(* PLC project PLCC Raw Material Accounting System, Machine Expert Logic Builder V23.0.22.0, author nikiden *)
(* stored: creationDateTime 2026-09-22T13:28:06.869679+00:00, version 0.0.0.0, modificationDateTime 2026-09-10T08:01:48.8091995, organization Briansk Cardboard *)

TYPE E_ChannelStatus :
(
    CHANNEL_STATUS_STARTING     := 0,    // Ожидание первого корректного отсчёта HSC.
    CHANNEL_STATUS_RUNNING      := 1,    // Канал работает штатно.
    CHANNEL_STATUS_HSC_INVALID  := 2,    // HSC временно не подтверждает достоверность данных.
    CHANNEL_STATUS_HSC_ERROR    := 3,    // Аппаратный HSC сообщил об ошибке.
    CHANNEL_STATUS_COUNTER_JUMP := 4,    // Обнаружен недопустимо большой скачок счётчика.
    CHANNEL_STATUS_CONFIG_ERROR := 5     // Ошибка настроек диапазона HSC или пересчёта.
);
END_TYPE

TYPE E_RollEndReason :
(
    ROLL_END_NONE   := 0,    // Рулон ещё не завершался.
    ROLL_END_SPLICE := 1,    // Рулон завершён кнопкой SPLICE.
    ROLL_END_RESET  := 2     // Рулон завершён ручной кнопкой RESET.
);
END_TYPE

TYPE ST_HscState :
STRUCT
    xInitialized         : BOOL;             // Получен первый корректный абсолютный отсчёт HSC.
    udiPreviousAbs       : UDINT;            // Абсолютное значение HSC на предыдущем цикле.
    udiPulseDelta        : UDINT;            // Число новых импульсов за текущий цикл ПЛК.
    xDataValid           : BOOL;             // Приращение импульсов разрешено использовать.
    xJumpDetected        : BOOL;             // Одноцикловый признак недопустимого скачка HSC.
    udiRejectedJumpCount : UDINT;            // Количество отброшенных скачков HSC.
    eStatus              : E_ChannelStatus;  // Текущее состояние канала.
END_STRUCT
END_TYPE

TYPE ST_LineState :
STRUCT
    uliTotalPulses   : ULINT;  // Общее число импульсов шестого энкодера после запуска ПЛК.
    uliTotalLengthMm : ULINT;  // Общий метраж линии в миллиметрах после запуска ПЛК.
    rSpeedMPerMin    : REAL;   // Текущая скорость линии в метрах в минуту.
    xMoving          : BOOL;   // TRUE, если за последний интервал пришли импульсы.
    xConfigFault     : BOOL;   // Ошибка параметров энкодера, колеса или интервала скорости.
END_STRUCT
END_TYPE

TYPE ST_RollEvent :
STRUCT
    udiEventId         : UDINT;          // Уникальный номер события; назначается постоянной очередью.
    udiTimestampUtc    : UDINT;          // UNIX-время завершения рулона в секундах UTC.
    usiUnwindNumber    : USINT;          // Постоянный физический номер раската 1...5.
    usiShiftNumber     : USINT;          // Номер смены, в которой завершился рулон: 1 или 2.
    eEndReason         : E_RollEndReason;// Причина завершения: SPLICE или допустимый RESET.
    udiLengthMm        : UDINT;          // Итоговая длина завершённого рулона в миллиметрах, максимум около 4295 км.
END_STRUCT
END_TYPE

TYPE ST_RollState :
STRUCT
    uliCurrentRollPulses       : ULINT;           // Накопленные импульсы текущего рулона.
    uliCurrentLengthMm         : ULINT;           // Длина текущего рулона в миллиметрах.
    uliPreviousRollPulses      : ULINT;           // Импульсы последнего учтённого рулона.
    uliPreviousRollLengthMm    : ULINT;           // Длина последнего учтённого рулона в миллиметрах.
    udiRollSequenceNumber      : UDINT;           // Порядковый номер текущего рулона внутри канала.
    eLastEndReason             : E_RollEndReason; // Причина завершения предыдущего учтённого рулона.
    xRollCompleted             : BOOL;            // Одноцикловый сигнал завершения учтённого рулона.
    xShortResetDiscarded       : BOOL;            // Одноцикловый сигнал RESET при длине менее 100 м.
    uliLastDiscardedLengthMm   : ULINT;           // Длина последнего отброшенного короткого рулона.
    uliDiscardedTotalLengthMm  : ULINT;           // Общая отброшенная длина после коротких RESET.
    xConfigFault               : BOOL;            // Ошибка параметров энкодера или мерного колеса.
END_STRUCT
END_TYPE

TYPE ST_ShiftState :
STRUCT
    usiCurrentShift : USINT;  // Номер текущей смены: 1 или 2.
    xRtcValid       : BOOL;   // RTC контроллера прочитан без ошибки.
    xShiftChanged   : BOOL;   // Одноцикловый признак смены номера смены.
    uiLocalHour     : UINT;   // Текущий местный час, 0...23.
    uiLocalMinute   : UINT;   // Текущая местная минута, 0...59.
    uiLocalSecond   : UINT;   // Текущая местная секунда, 0...59.
    uiLocalYear     : UINT;   // Год местного времени, например 2026.
    uiLocalMonth    : UINT;   // Месяц местного времени, 1...12.
    uiLocalDay      : UINT;   // День месяца местного времени, 1...31.
    udiTimestampUtc : UDINT;  // Текущее UNIX-время в секундах UTC для отметки событий.
    udiRtcError     : UDINT;  // Код ошибки функции чтения RTC, 0 означает отсутствие ошибки.
END_STRUCT
END_TYPE

TYPE ST_StopJournalEvent :
STRUCT
    udiEventId                  : UDINT; // Постоянный ID события линии ЛГК.
    udiTimestampUtc             : UDINT; // UNIX UTC; 0, если RTC неисправен.
    wKind                       : WORD;  // 1=состояние, 2=завершение смены, 3=новый заказ.
    wStateCode                  : WORD;  // Старые коды ProductionLine; 32768=граница смены.
    wShiftNumber                : WORD;  // Смена, к которой относится снимок.
    udiOrderNumber              : UDINT; // Номер заказа на момент события.
    udiOrderLengthDm            : UDINT; // Метраж заказа, 0,1 м.
    udiOrderAreaX100            : UDINT; // Площадь заказа, м2 x 100.
    udiShiftLengthDm            : UDINT; // Метраж смены, 0,1 м.
    udiShiftAreaX100            : UDINT; // Площадь смены, м2 x 100.
    wSpeedDmPerMin              : WORD;  // Скорость, 0,1 м/мин.
    wOperatorNumber             : WORD;  // Номер оператора.
    wChangeoverSetpointTenthsMin: WORD;  // Норматив переналадки, 0,1 мин.
    wAlarmBits                  : WORD;  // Диагностика нового ПЛК; не старый Status2.
    wBreakPoint                 : WORD;  // Точка обрыва 1...5.
    wBreakSide                  : WORD;  // Сторона обрыва 1...2.
    wBreakReason                : WORD;  // Причина обрыва 1...3.
END_STRUCT
END_TYPE

TYPE ST_StopJournalPersistent :
STRUCT
    a_stQueue        : ARRAY[0..127] OF ST_StopJournalEvent;
    uiHead           : UINT;
    uiTail           : UINT;
    uiCount          : UINT;
    udiNextEventId   : UDINT;
    udiOverflowCount : UDINT;
    uliLinePulses    : ULINT;
    wLastState       : WORD;
    dwSignature      : DWORD;
END_STRUCT
END_TYPE

TYPE ST_StopMachinePersistent :
STRUCT
    wConfigSignature                 : WORD;  // Сигнатура инициализированных постоянных настроек.
    udiOrderNumber                   : UDINT; // Номер заказа, показываемый оператору.
    udiOrderDatabaseId               : UDINT; // NumZ: ключ записи заказа в БД.
    udiOrderTechnicalCard            : UDINT; // NumTK: номер технологической карты.
    uiOrderSourceShift               : UINT;  // NumSM, полученный с сервера.
    uiOrderNominalSpeed              : UINT;  // Efficiency из записи заказа.
    uiOperatorNumber                 : UINT;  // Номер авторизованного оператора будущей EB-панели.
    wLastServerOrderSequence         : WORD;  // Последний атомарно применённый пакет сервера.
    uliOrderBaselineMm               : ULINT; // Общий метраж линии в момент начала заказа.
    uliShiftBaselineMm               : ULINT; // Общий метраж линии в момент начала смены.
    uiAreaCoefficientX100            : UINT;  // Площадь на метр, м2/м x 100 (210 = 2,10).
    uiStartDetectLengthDm            : UINT;  // Путь подтверждения работы, 0,1 м.
    uiChangeoverSetpointTenthsMin    : UINT;  // Допустимая переналадка, 0,1 мин.
    usiLastShiftNumber               : USINT; // Последняя смена для восстановления после отключения.
END_STRUCT
END_TYPE

TYPE ST_StopMachineState :
STRUCT
    wStateCode                         : WORD;  // Текущее состояние ЛГК по таблице состояний.
    wStatusBits                        : WORD;  // Диагностические признаки интерфейса Стопмашины.
    wAlarmBits                         : WORD;  // Активные предупреждения интерфейса.
    udiOrderNumber                     : UDINT; // Номер текущего заказа.
    udiOrderDatabaseId                 : UDINT; // Ключ текущего заказа в БД.
    udiOrderTechnicalCard              : UDINT; // Номер технологической карты.
    uiOrderSourceShift                 : UINT;  // Номер смены из записи заказа сервера.
    uiOrderNominalSpeed                : UINT;  // Номинальная скорость из записи заказа.
    uiOperatorNumber                   : UINT;  // Номер оператора EB-панели.
    udiCurrentOrderLengthDm            : UDINT; // Выпуск текущего заказа, 0,1 м.
    udiShiftLengthDm                   : UDINT; // Выпуск текущей смены, 0,1 м.
    udiCurrentOrderAreaX100            : UDINT; // Площадь текущего заказа, м2 x 100.
    udiShiftAreaX100                   : UDINT; // Площадь текущей смены, м2 x 100.
    uiSpeedDmPerMin                    : UINT;  // Скорость, 0,1 м/мин.
    uiChangeoverRemainingTenthsMin     : UINT;  // Остаток переналадки, 0,1 мин.
    usiLastBreakPoint                  : USINT; // Последняя точка обрыва: 1...5.
    usiLastBreakSide                   : USINT; // Сторона: 1 верх, 2 низ.
    usiLastBreakReason                 : USINT; // Причина: 1 сырьё, 2 оборудование, 3 машинист.
    wLastCommandResult                 : WORD;  // Результат последней обработанной команды HMI.
    wLastProcessedSequence             : WORD;  // Последовательность последней команды HMI.
    wLastServerOrderResult              : WORD;  // Результат обработки последнего пакета заказа.
    wLastServerOrderSequence            : WORD;  // Последовательность последнего пакета заказа.
    xPackingComplete                   : BOOL;  // Оператор подтвердил завершение упаковки.
    xChangeoverOverdue                 : BOOL;  // Превышено заданное время переналадки.
    xCommandRejected                   : BOOL;  // Последняя полученная команда отклонена.
    xConfigFault                       : BOOL;  // Некорректные сохранённые настройки.
    xServerOrderValid                  : BOOL;  // PLC получил корректный заказ от сервера.
    xInitialized                       : BOOL;  // Блок прошёл первичную инициализацию.
END_STRUCT
END_TYPE

TYPE ST_SystemDiagnostics :
STRUCT
    a_eHscStatus      : ARRAY[1..6] OF E_ChannelStatus; // Состояния шести каналов HSC.
    a_xHscFault       : ARRAY[1..6] OF BOOL;            // Ошибка соответствующего канала HSC.
    a_xHmiOverflow    : ARRAY[1..5] OF BOOL;            // Значение канала не помещается в 32 бита DWIN.
    xAnyHscFault      : BOOL;                           // Есть хотя бы одна ошибка HSC.
    xAnyConfigFault   : BOOL;                           // Есть ошибка параметров пересчёта.
    xRtcFault         : BOOL;                           // Не удалось получить время контроллера.
    uliProgramCycles  : ULINT;                          // Счётчик циклов SR_Main для диагностики.
END_STRUCT
END_TYPE

(* global variable list GVL_Constants *)
VAR_GLOBAL CONSTANT
    c_iRollChannelCount              : INT   := 5;                    // Количество раскатов сырья.
    c_iHscChannelCount               : INT   := 6;                    // Пять раскатов и один энкодер линии.
    c_udiEncoderPulsesPerRevolution  : UDINT := UDINT#250;            // Импульсов энкодера за один оборот.
    c_udiWheelCircumferenceMm        : UDINT := UDINT#250;            // Окружность каждого мерного колеса, мм.
    c_udiHscCounterRange             : UDINT := UDINT#1000000000;     // Диапазон HSC: значения 0...999999999.
    c_udiMaxPulseDeltaPerCycle       : UDINT := UDINT#100000;         // Защита от ложного скачка или сброса HSC.
    c_tInputFilter                   : TIME  := T#50ms;                // Время подтверждения нажатия кнопки.
    c_uliManualResetMinLengthMm      : ULINT := ULINT#100000;         // Минимум 100 м для учёта ручного RESET.
    c_tSpeedSample                   : TIME  := T#1s;                  // Интервал обновления скорости линии.
    c_tHaiwellActivityHold           : TIME  := T#10s;                 // Удержание признака движения для медленного опроса HMI.
    c_tHaiwellFlashHalfPeriod        : TIME  := T#250ms;               // Три быстрые жёлтые вспышки: 0,25 с ВКЛ и 0,25 с ВЫКЛ.
    c_tHaiwellResetHold              : TIME  := T#3s;                  // Время показа состояния RESET на центральной HMI.
    c_usiShift_1_StartHour           : USINT := USINT#8;              // Начало первой смены, 08:00.
    c_usiShift_2_StartHour           : USINT := USINT#20;             // Начало второй смены, 20:00.
    c_udiShiftMaxIntervalSeconds     : UDINT := UDINT#43200;          // Максимум одного сменного интервала: 12 часов.
    c_udiLocalUtcOffsetSeconds       : UDINT := UDINT#10800;          // Брянск: UTC+3, то есть 3 часа.
    c_dwPersistentLayoutSignature    : DWORD := DWORD#16#4342504C;    // ASCII "CBPL": признак нашей структуры PERSISTENT.
    c_wPersistentLayoutVersion       : WORD  := WORD#2;                // Версия разметки постоянной памяти.
    c_wHaiwellProtocolVersion        : WORD  := WORD#2;                // Версия read-only карты центральной Haiwell.

    // Отдельный интерфейс Стопмашины ЛГК. Он не содержит номера линии.
    c_wStopMachineSignature          : WORD  := WORD#16#534D;         // ASCII "SM".
    c_wStopMachineProtocolVersion    : WORD  := WORD#2;
    c_wServerOrderApplyCommand       : WORD  := WORD#16#4F52;         // ASCII "OR": применить пакет заказа сервера.
    c_uiStopDefaultAreaCoefficientX100 : UINT := UINT#210;            // 2,10 м2 на метр.
    c_uiStopDefaultStartDetectLengthDm : UINT := UINT#500;            // 50,0 м.
    c_uiStopDefaultChangeoverTenthsMin : UINT := UINT#0;              // Таймер отключён до настройки.
    c_tStopNoFeedDelay               : TIME  := T#20s;

    c_wStopStateRunning              : WORD := WORD#1;
    c_wStopStateStopped              : WORD := WORD#2;
    c_wStopStateNoFeed               : WORD := WORD#8;
    c_wStopStateChangeover           : WORD := WORD#16;
    c_wStopStateProduction           : WORD := WORD#32;
    c_wStopStatePpr                  : WORD := WORD#64;
    c_wStopStateLunch                : WORD := WORD#128;
    c_wStopStateRepair               : WORD := WORD#256;
    c_wStopStateAlarm                : WORD := WORD#512;
    c_wStopStateTechnology           : WORD := WORD#1024;
    c_wStopStateBreak                : WORD := WORD#2048;

    c_wStopCommandStop               : WORD := WORD#1;
    c_wStopCommandStart              : WORD := WORD#2;
    c_wStopCommandChangeover         : WORD := WORD#3;
    c_wStopCommandProduction         : WORD := WORD#4;
    c_wStopCommandLunch              : WORD := WORD#5;
    c_wStopCommandPpr                : WORD := WORD#6;
    c_wStopCommandRepair             : WORD := WORD#7;
    c_wStopCommandAlarm              : WORD := WORD#8;
    c_wStopCommandTechnology         : WORD := WORD#9;
    c_wStopCommandBreak              : WORD := WORD#10;
    c_wStopCommandPackingComplete    : WORD := WORD#11;
    c_wStopCommandSetOperator        : WORD := WORD#12;
    c_wStopCommandApplySettings      : WORD := WORD#20;

    c_wStopResultNone                : WORD := WORD#0;
    c_wStopResultAccepted            : WORD := WORD#1;
    c_wStopResultInvalidCode         : WORD := WORD#2;
    c_wStopResultInvalidParameter    : WORD := WORD#3;
    c_wStopResultInvalidState        : WORD := WORD#4;                // Команда состояния противоречит движению энкодера.
END_VAR

(* global variable list GVL_IO *)
VAR_GLOBAL
    udiHscAbs : ARRAY[1..6] OF UDINT; // Абсолютные показания шести аппаратных HSC.
    xHscValid : ARRAY[1..6] OF BOOL;  // Достоверность выходов соответствующего HSC.
    xHscError : ARRAY[1..6] OF BOOL;  // Ошибка соответствующего аппаратного HSC.
    xReset    : ARRAY[1..5] OF BOOL;  // Кнопки RESET раскатов 1...5 с TM3DI16, входы I0...I4.
    xSplice   : ARRAY[1..5] OF BOOL;  // Кнопки SPLICE раскатов 1...5 с TM3DI16, входы I5...I9.
END_VAR

(* global variable list GVL_Runtime *)
VAR_GLOBAL
    a_stHscState  : ARRAY[1..6] OF ST_HscState;  // Рабочее состояние шести каналов HSC.
    stLineState   : ST_LineState;                // Скорость и общий метраж шестого энкодера.
    stShiftState  : ST_ShiftState;               // Номер смены и состояние часов контроллера.
    stStopMachine : ST_StopMachineState;         // Изолированное состояние Стопмашины линии ЛГК.
END_VAR

(* global variable list GVL_HMI *)
VAR_GLOBAL
    a_wHmi1Tx : ARRAY[0..12] OF WORD; // Регистры VP 2000...200C панели раската №1.
    a_wHmi2Tx : ARRAY[0..12] OF WORD; // Регистры VP 2000...200C панели раската №2.
    a_wHmi3Tx : ARRAY[0..12] OF WORD; // Регистры VP 2000...200C панели раската №3.
    a_wHmi4Tx : ARRAY[0..12] OF WORD; // Регистры VP 2000...200C панели раската №4.
    a_wHmi5Tx : ARRAY[0..12] OF WORD; // Регистры VP 2000...200C панели раската №5.

    // Системный пакет установки встроенных часов DWIN через VP 009C...009F.
    a_wHmi1RtcSync : ARRAY[0..3] OF WORD;
    a_wHmi2RtcSync : ARRAY[0..3] OF WORD;
    a_wHmi3RtcSync : ARRAY[0..3] OF WORD;
    a_wHmi4RtcSync : ARRAY[0..3] OF WORD;
    a_wHmi5RtcSync : ARRAY[0..3] OF WORD;
END_VAR

(* global variable list GVL_Diagnostics *)
VAR_GLOBAL
    stSystem : ST_SystemDiagnostics; // Общая диагностика проекта для онлайн-контроля и будущей SCADA.
END_VAR

(* global variable list PersistentVars *)
VAR_GLOBAL PERSISTENT RETAIN
    a_stEventQueue       : ARRAY[0..127] OF ST_RollEvent; // Постоянная кольцевая очередь на 128 событий.
    uiEventQueueHead     : UINT := UINT#0;                // Индекс первого события, ожидающего подтверждения.
    uiEventQueueTail     : UINT := UINT#0;                // Индекс ячейки для записи следующего события.
    uiEventQueueCount    : UINT := UINT#0;                // Текущее количество событий в очереди.
    udiNextEventId       : UDINT := UDINT#1;              // Уникальный номер, который получит следующее событие.
    udiQueueOverflowCount: UDINT := UDINT#0;              // Число событий, не помещённых из-за полной очереди.
    a_stRollState        : ARRAY[1..5] OF ST_RollState;   // Сохраняемое состояние текущего и предыдущего рулона каждого раската.
    stStopMachine        : ST_StopMachinePersistent;      // Заказ, базовые метражи и настройки Стопмашины ЛГК.
    usiShiftAccumulatorNumber : USINT;                    // Смена, к которой относятся накопители центральной HMI.
    udiShiftStartTimestampUtc : UDINT;                    // UTC-время начала текущего интервала накопления.
    a_uliShiftRollPulses : ARRAY[1..5] OF ULINT;           // Импульсы каждого раската с начала текущей смены.
    uliShiftOutputPulses : ULINT;                          // Импульсы шестого энкодера с начала текущей смены.
    dwLayoutSignature    : DWORD;                          // Сигнатура разметки; ноль или несовпадение запускает безопасную инициализацию.
    wLayoutVersion       : WORD;                           // Версия разметки постоянной памяти.
    stStopJournal        : ST_StopJournalPersistent;       // Независимая очередь событий ЛГК; добавлена в конец разметки.
END_VAR

(* global variable list GVL_SCADA *)
VAR_GLOBAL
    a_wEventPacket AT %MW2000 : ARRAY[0..11] OF WORD; // Событие протокола v2: 12 последовательных слов.
    wEventReady AT %MW2012 : WORD;                    // 1 — пакет содержит событие, 0 — очередь пуста.
    wQueueCount AT %MW2013 : WORD;                    // Количество неподтверждённых событий в очереди.
    wQueueCapacity AT %MW2014 : WORD;                 // Полная ёмкость очереди, сейчас 128 событий.
    wQueueStatus AT %MW2015 : WORD;                   // 0 — пусто, 1 — есть данные, 2 — заполнена, 3 — ошибка хранилища, 4 — исчерпан EventId.

    a_wAckEventId AT %MW2016 : ARRAY[0..1] OF WORD;   // EventId UDINT, подтверждаемый сервером; старшее слово первым.
    wAckCommand AT %MW2018 : WORD;                    // Сервер записывает 16#A55A после сохранения события на диск.
    wCollectorHeartbeat AT %MW2019 : WORD;            // Счётчик жизни службы-сборщика; записывается сервером.
    wLastAckResult AT %MW2020 : WORD;                 // 0 — подтверждений не было, 1 — принято, 2 — отклонено.
    a_wQueueOverflowCount AT %MW2021 : ARRAY[0..1] OF WORD; // Число событий, отвергнутых из-за полной очереди.

    // Сервер -> PLC: новый заказ ЛГК. Параметры и sequence записываются первыми,
    // wOrderCommand = 16#4F52 записывается последним. PLC очищает команду сам.
    wOrderCommand AT %MW2030 : WORD;
    wOrderSequence AT %MW2031 : WORD;
    a_wOrderDatabaseId AT %MW2032 : ARRAY[0..1] OF WORD;     // NumZ из ExternalProductionData, старшее слово первым.
    a_wOrderTechnicalCard AT %MW2034 : ARRAY[0..1] OF WORD;  // NumTK, старшее слово первым.
    a_wOrderDisplayNumber AT %MW2036 : ARRAY[0..1] OF WORD;  // Числовая часть Zakaz для экрана, старшее слово первым.
    wOrderSourceShift AT %MW2038 : WORD;                     // NumSM от сервера.
    wOrderNominalSpeed AT %MW2039 : WORD;                    // Efficiency, единицы исходной БД.
    wOrderChangeoverTenthsMin AT %MW2040 : WORD;             // ReconfigurationT x 10.

    // PLC -> сервер: результат применения заказа.
    wOrderApplyResult AT %MW2041 : WORD;                     // 0 — нет, 1 — принят, 2 — неверная команда, 3 — неверные данные.
    wLastOrderSequence AT %MW2042 : WORD;
END_VAR

(* global variable list GVL_HAIWELL *)
VAR_GLOBAL
    // Непрерывная read-only область Modbus TCP для центральной Haiwell A10-W.
    // Многословные значения передаются в порядке: старшее WORD, затем младшее WORD.

    wHmiSignature       AT %MW2100 : WORD; // 16#484D ('HM').
    wHmiProtocolVersion AT %MW2101 : WORD; // Версия карты.
    wPlcHeartbeat       AT %MW2102 : WORD; // Изменяется раз в секунду.
    wSystemStatusBits   AT %MW2103 : WORD; // Общие диагностические флаги.
    wCurrentShift       AT %MW2104 : WORD; // 1, 2 или 0 при недостоверном RTC.
    wLocalHour          AT %MW2105 : WORD; // 0...23.
    wLocalMinute        AT %MW2106 : WORD; // 0...59.
    wEventQueueCount    AT %MW2107 : WORD;
    wEventQueueStatus   AT %MW2108 : WORD;
    wLastAckResult      AT %MW2109 : WORD;

    a_wCurrentLengthX10  AT %MW2110 : ARRAY[1..5, 0..1] OF WORD;
    a_wPreviousLengthX10 AT %MW2120 : ARRAY[1..5, 0..1] OF WORD;
    a_wUnwindStatus      AT %MW2130 : ARRAY[1..5] OF WORD;
    a_wLastEndReason     AT %MW2135 : ARRAY[1..5] OF WORD;

    a_wOutputTotalLengthX10 AT %MW2140 : ARRAY[0..1] OF WORD;
    wOutputSpeedX10         AT %MW2142 : WORD;
    wOutputStatus           AT %MW2143 : WORD;
    a_wDiscardedLengthX10   AT %MW2144 : ARRAY[1..5, 0..1] OF WORD;
    a_wQueueOverflowCount   AT %MW2154 : ARRAY[0..1] OF WORD;
    wCollectorHeartbeat     AT %MW2156 : WORD;
    wReserved2157           AT %MW2157 : WORD;

    // Состояния, дата и накопители текущей смены.
    a_wUnwindDisplayState       AT %MW2200 : ARRAY[1..5] OF WORD;    // 0 — стоит, 1 — работает, 2 — жёлтая фаза SPLICE/RESET.
    wLocalYear                  AT %MW2205 : WORD;
    wLocalMonth                 AT %MW2206 : WORD;
    wLocalDay                   AT %MW2207 : WORD;
    a_wReserved2208             AT %MW2208 : ARRAY[0..1] OF WORD;
    a_wShiftOutputLengthX10     AT %MW2210 : ARRAY[0..1] OF WORD;
    wShiftAverageSpeedX10       AT %MW2212 : WORD;
    wShiftStatus                AT %MW2213 : WORD;                   // bit 0 — накопители достоверны.
    a_wShiftRollLengthX10       AT %MW2214 : ARRAY[1..5, 0..1] OF WORD;
    a_wShiftRawTotalLengthX10   AT %MW2224 : ARRAY[0..1] OF WORD;
    a_wReserved2226             AT %MW2226 : ARRAY[0..3] OF WORD;
END_VAR

(* global variable list GVL_StopMachine *)
VAR_GLOBAL
    // ========================================================
    // PLC -> HMI. Только чтение со стороны панели, MW2300...2359
    // ========================================================
    wSignature AT %MW2300 : WORD;
    wProtocolVersion AT %MW2301 : WORD;
    wPlcHeartbeat AT %MW2302 : WORD;
    wStateCode AT %MW2303 : WORD;
    wStatusBits AT %MW2304 : WORD;
    wAlarmBits AT %MW2305 : WORD;
    wShiftNumber AT %MW2306 : WORD;
    wLocalHour AT %MW2307 : WORD;
    wLocalMinute AT %MW2308 : WORD;
    wLocalSecond AT %MW2309 : WORD;
    a_wOrderNumber AT %MW2310 : ARRAY[0..1] OF WORD;
    a_wOrderLengthDm AT %MW2312 : ARRAY[0..1] OF WORD;
    a_wOrderAreaX100 AT %MW2314 : ARRAY[0..1] OF WORD;
    a_wShiftLengthDm AT %MW2316 : ARRAY[0..1] OF WORD;
    a_wShiftAreaX100 AT %MW2318 : ARRAY[0..1] OF WORD;
    wSpeedDmPerMin AT %MW2320 : WORD;
    wChangeoverRemainingTenthsMin AT %MW2321 : WORD;
    wChangeoverSetpointTenthsMin AT %MW2322 : WORD;
    wStartDetectLengthDm AT %MW2323 : WORD;
    wAreaCoefficientX100 AT %MW2324 : WORD;
    wLastBreakPoint AT %MW2325 : WORD;
    wLastBreakSide AT %MW2326 : WORD;
    wLastBreakReason AT %MW2327 : WORD;
    wPackingComplete AT %MW2328 : WORD;
    wLastCommandResult AT %MW2329 : WORD;
    wLastProcessedSequence AT %MW2330 : WORD;
    wPhysicalControlEnabled AT %MW2331 : WORD; // Всегда 0: HMI не управляет оборудованием.
    a_wOrderDatabaseId AT %MW2332 : ARRAY[0..1] OF WORD;
    a_wOrderTechnicalCard AT %MW2334 : ARRAY[0..1] OF WORD;
    wOrderSourceShift AT %MW2336 : WORD;
    wOrderNominalSpeed AT %MW2337 : WORD;
    wOperatorNumber AT %MW2338 : WORD;
    a_wReservedRead AT %MW2339 : ARRAY[0..20] OF WORD;

    // ========================================================
    // HMI -> PLC. Панель пишет только MW2360...2399
    // Команда передаётся последней; sequence меняется для каждого действия.
    // ========================================================
    wCommandCode AT %MW2360 : WORD;
    wCommandSequence AT %MW2361 : WORD;
    wCommandParam0 AT %MW2362 : WORD;
    wCommandParam1 AT %MW2363 : WORD;
    wCommandParam2 AT %MW2364 : WORD;
    wSettingStartDetectLengthDm AT %MW2365 : WORD;
    wSettingAreaCoefficientX100 AT %MW2366 : WORD;
    wSettingChangeoverTenthsMin AT %MW2367 : WORD;
    wHmiHeartbeat AT %MW2368 : WORD;
    a_wReservedWrite AT %MW2369 : ARRAY[0..30] OF WORD;
END_VAR

(* global variable list GVL_StopJournal *)
VAR_GLOBAL
    // Снимок первого события. PLC -> сервер, 2400...2422.
    wSignature AT %MW2400 : WORD;                 // 16#534A = SJ.
    wVersion AT %MW2401 : WORD;                   // Версия протокола 1.
    a_wEventId AT %MW2402 : ARRAY[0..1] OF WORD; // Старшее слово первым.
    a_wTimestampUtc AT %MW2404 : ARRAY[0..1] OF WORD;
    wKind AT %MW2406 : WORD;
    wStateCode AT %MW2407 : WORD;
    wShiftNumber AT %MW2408 : WORD;
    a_wOrderNumber AT %MW2409 : ARRAY[0..1] OF WORD;
    a_wOrderLengthDm AT %MW2411 : ARRAY[0..1] OF WORD;
    a_wOrderAreaX100 AT %MW2413 : ARRAY[0..1] OF WORD;
    wSpeedDmPerMin AT %MW2415 : WORD;
    wOperatorNumber AT %MW2416 : WORD;
    wChangeoverSetpointTenthsMin AT %MW2417 : WORD;
    wAlarmBits AT %MW2418 : WORD;
    wBreakPoint AT %MW2419 : WORD;
    wBreakSide AT %MW2420 : WORD;
    wBreakReason AT %MW2421 : WORD;
    a_wShiftLengthDm AT %MW2422 : ARRAY[0..1] OF WORD;
    a_wShiftAreaX100 AT %MW2424 : ARRAY[0..1] OF WORD;
    wEventReady AT %MW2426 : WORD;
    wQueueCount AT %MW2427 : WORD;
    wQueueStatus AT %MW2428 : WORD;               // 0=норма, 1=полна, 2=переполнение, 3=повреждение, 4=ID исчерпан.
    // Сервер -> PLC: ID записать первым, команду 16#A55B — последней.
    a_wAckEventId AT %MW2429 : ARRAY[0..1] OF WORD;
    wAckCommand AT %MW2431 : WORD;
    wLastAckResult AT %MW2432 : WORD;             // 0=нет, 1=принят, 2=отклонён.
    a_wOverflowCount AT %MW2433 : ARRAY[0..1] OF WORD;
    wHeartbeat AT %MW2435 : WORD;
    a_wReserved AT %MW2436 : ARRAY[0..23] OF WORD;
END_VAR

FUNCTION_BLOCK FB_DwinDataPacker
VAR_INPUT
    i_uliCurrentLengthMm  : ULINT; // Текущая длина рулона в миллиметрах.
    i_uliPreviousLengthMm : ULINT; // Предыдущая длина рулона в миллиметрах.
    i_usiUnwindNumber     : USINT; // Постоянный физический номер раската 1...5.
END_VAR

VAR_OUTPUT
    q_wCurrentHigh  : WORD; // VP 2000: старшее слово текущей длины.
    q_wCurrentLow   : WORD; // VP 2001: младшее слово текущей длины.
    q_wPreviousHigh : WORD; // VP 2002: старшее слово предыдущей длины.
    q_wPreviousLow  : WORD; // VP 2003: младшее слово предыдущей длины.
    q_wUnwindNumber : WORD; // VP 2004: постоянный физический номер раската.
    q_xOverflow     : BOOL; // Одно из значений превысило диапазон 32-битного DWIN.
END_VAR

VAR
    uliCurrentX10  : ULINT; // Текущая длина в десятых долях метра.
    uliPreviousX10 : ULINT; // Предыдущая длина в десятых долях метра.
    udiCurrentX10  : UDINT; // Ограниченное 32-битное значение текущей длины.
    udiPreviousX10 : UDINT; // Ограниченное 32-битное значение предыдущей длины.
END_VAR

VAR CONSTANT
    c_uliDwinMaxValue : ULINT := ULINT#4294967295; // Максимум Unsigned Long Int DWIN.
END_VAR

            // 100 мм соответствуют 0.1 м на экране DWIN.
uliCurrentX10 := i_uliCurrentLengthMm / ULINT#100;
uliPreviousX10 := i_uliPreviousLengthMm / ULINT#100;
IF (i_uliPreviousLengthMm MOD ULINT#100) >= ULINT#50 THEN
    uliPreviousX10 := uliPreviousX10 + ULINT#1;
END_IF;
q_xOverflow := FALSE;


IF uliCurrentX10 > c_uliDwinMaxValue THEN
    udiCurrentX10 := UDINT#4294967295;
    q_xOverflow := TRUE;
ELSE
    udiCurrentX10 := ULINT_TO_UDINT(uliCurrentX10);
END_IF;


IF uliPreviousX10 > c_uliDwinMaxValue THEN
    udiPreviousX10 := UDINT#4294967295;
    q_xOverflow := TRUE;
ELSE
    udiPreviousX10 := ULINT_TO_UDINT(uliPreviousX10);
END_IF;


q_wCurrentHigh :=
    UDINT_TO_WORD(udiCurrentX10 / UDINT#65536);

q_wCurrentLow :=
    UDINT_TO_WORD(udiCurrentX10 MOD UDINT#65536);

q_wPreviousHigh :=
    UDINT_TO_WORD(udiPreviousX10 / UDINT#65536);

q_wPreviousLow :=
    UDINT_TO_WORD(udiPreviousX10 MOD UDINT#65536);

q_wUnwindNumber := USINT_TO_WORD(i_usiUnwindNumber);

          
END_FUNCTION_BLOCK

FUNCTION_BLOCK FB_EventPacker
VAR_INPUT
    i_xEventValid : BOOL;         // TRUE — входная структура содержит событие для передачи.
    i_stEvent     : ST_RollEvent; // Первое неподтверждённое событие постоянной очереди.
END_VAR

VAR_OUTPUT
    q_a_wPacket   : ARRAY[0..11] OF WORD; // Пакет протокола v2: 12 слов, старшие слова идут первыми.
    q_xPacketValid: BOOL;                 // TRUE — пакет заполнен и CRC рассчитан.
END_VAR

VAR
    iWord       : INT;  // Индекс слова при очистке пакета и вычислении CRC.
    iByte       : INT;  // Индекс байта внутри слова: сначала старший, затем младший.
    iBit        : INT;  // Индекс бита при вычислении CRC16 Modbus.
    wCrc        : WORD; // Рабочее значение CRC16 Modbus.
    wSourceWord : WORD; // Текущее слово пакета, участвующее в CRC.
    byData      : BYTE; // Текущий байт пакета, участвующий в CRC.
END_VAR

VAR CONSTANT
    c_wSignature      : WORD := WORD#16#CB01; // Сигнатура протокола CBPL, защищает от неверного разбора пакета.
    c_wProtocolVersion: WORD := WORD#2;       // Версия 2: EventId и длина передаются как UDINT.
END_VAR

            q_xPacketValid := FALSE;

FOR iWord := 0 TO 11 DO
    q_a_wPacket[iWord] := WORD#0;
END_FOR;


IF i_xEventValid THEN

    // 0: сигнатура; 1: версия протокола.
    q_a_wPacket[0] := c_wSignature;
    q_a_wPacket[1] := c_wProtocolVersion;

    // 2...3: EventId UDINT, старшее слово идёт первым.
    q_a_wPacket[2] := UDINT_TO_WORD(i_stEvent.udiEventId / UDINT#65536);
    q_a_wPacket[3] := UDINT_TO_WORD(i_stEvent.udiEventId MOD UDINT#65536);

    // 4...5: UNIX-время UTC UDINT, старшее слово идёт первым.
    q_a_wPacket[4] := UDINT_TO_WORD(i_stEvent.udiTimestampUtc / UDINT#65536);
    q_a_wPacket[5] := UDINT_TO_WORD(i_stEvent.udiTimestampUtc MOD UDINT#65536);

    // 6...8: физический раскат, смена и причина передаются отдельными словами.
    q_a_wPacket[6] := USINT_TO_WORD(i_stEvent.usiUnwindNumber);
    q_a_wPacket[7] := USINT_TO_WORD(i_stEvent.usiShiftNumber);

    CASE i_stEvent.eEndReason OF
        ROLL_END_SPLICE:
            q_a_wPacket[8] := WORD#1;
        ROLL_END_RESET:
            q_a_wPacket[8] := WORD#2;
        ELSE
            q_a_wPacket[8] := WORD#0;
    END_CASE;

    // 9...10: длина завершённого рулона в миллиметрах, UDINT.
    q_a_wPacket[9] := UDINT_TO_WORD(i_stEvent.udiLengthMm / UDINT#65536);
    q_a_wPacket[10] := UDINT_TO_WORD(i_stEvent.udiLengthMm MOD UDINT#65536);


    // CRC16 Modbus по словам 0...10. В каждом слове сначала обрабатывается старший байт.
    wCrc := WORD#16#FFFF;

    FOR iWord := 0 TO 10 DO

        wSourceWord := q_a_wPacket[iWord];

        FOR iByte := 0 TO 1 DO

            IF iByte = 0 THEN
                byData := WORD_TO_BYTE(SHR(wSourceWord, 8));
            ELSE
                byData := WORD_TO_BYTE(wSourceWord AND WORD#16#00FF);
            END_IF;

            wCrc := wCrc XOR BYTE_TO_WORD(byData);

            FOR iBit := 0 TO 7 DO
                IF (wCrc AND WORD#1) <> WORD#0 THEN
                    wCrc := SHR(wCrc, 1) XOR WORD#16#A001;
                ELSE
                    wCrc := SHR(wCrc, 1);
                END_IF;
            END_FOR;

        END_FOR;

    END_FOR;

    q_a_wPacket[11] := wCrc;
    q_xPacketValid := TRUE;

END_IF;

          
END_FUNCTION_BLOCK

FUNCTION_BLOCK FB_HscTracker
VAR_INPUT
    i_udiHscAbs             : UDINT; // Текущее абсолютное значение аппаратного HSC.
    i_xHscValid             : BOOL;  // TRUE, если HSC подтверждает достоверность значения.
    i_xHscError             : BOOL;  // TRUE, если аппаратный HSC сообщил об ошибке.
    i_udiCounterRange       : UDINT; // Число значений HSC до перехода через ноль.
    i_udiMaxDeltaPerCycle   : UDINT; // Максимально допустимое приращение за цикл ПЛК.
END_VAR

VAR_IN_OUT
    iq_stState : ST_HscState; // Рабочее состояние конкретного канала HSC.
END_VAR

VAR
    uliCalculatedDelta : ULINT; // Промежуточное приращение без риска переполнения.
END_VAR

            // Одноцикловые и расчётные поля сначала сбрасываются.
iq_stState.udiPulseDelta := UDINT#0;
iq_stState.xDataValid := FALSE;
iq_stState.xJumpDetected := FALSE;
uliCalculatedDelta := ULINT#0;


// Проверяем параметры самого трекера.
IF (i_udiCounterRange = UDINT#0)
   OR (i_udiMaxDeltaPerCycle = UDINT#0) THEN

    iq_stState.eStatus := CHANNEL_STATUS_CONFIG_ERROR;


// Ошибка HSC имеет приоритет над признаком Validity.
ELSIF i_xHscError THEN

    iq_stState.eStatus := CHANNEL_STATUS_HSC_ERROR;


ELSIF NOT i_xHscValid THEN

    iq_stState.eStatus := CHANNEL_STATUS_HSC_INVALID;


// Первый исправный отсчёт используется только как начальная точка.
ELSIF NOT iq_stState.xInitialized THEN

    iq_stState.udiPreviousAbs := i_udiHscAbs;
    iq_stState.xInitialized := TRUE;
    iq_stState.xDataValid := TRUE;
    iq_stState.eStatus := CHANNEL_STATUS_RUNNING;


ELSE

    // Обычное приращение без перехода HSC через ноль.
    IF i_udiHscAbs >= iq_stState.udiPreviousAbs THEN

        uliCalculatedDelta :=
            UDINT_TO_ULINT(i_udiHscAbs)
            - UDINT_TO_ULINT(iq_stState.udiPreviousAbs);


    // Переход через заданный диапазон HSC.
    ELSIF iq_stState.udiPreviousAbs < i_udiCounterRange THEN

        uliCalculatedDelta :=
            (
                UDINT_TO_ULINT(i_udiCounterRange)
                - UDINT_TO_ULINT(iq_stState.udiPreviousAbs)
            )
            + UDINT_TO_ULINT(i_udiHscAbs);


    // Значение не соответствует настроенному диапазону.
    ELSE

        uliCalculatedDelta :=
            UDINT_TO_ULINT(i_udiMaxDeltaPerCycle) + ULINT#1;

    END_IF;


    // Запоминаем текущий абсолютный отсчёт как базу следующего цикла.
    iq_stState.udiPreviousAbs := i_udiHscAbs;


    // Реалистичное приращение разрешается использовать дальше.
    IF uliCalculatedDelta <= UDINT_TO_ULINT(i_udiMaxDeltaPerCycle) THEN

        iq_stState.udiPulseDelta :=
            ULINT_TO_UDINT(uliCalculatedDelta);

        iq_stState.xDataValid := TRUE;
        iq_stState.eStatus := CHANNEL_STATUS_RUNNING;


    // Огромный скачок отбрасывается и не попадает в метраж.
    ELSE

        iq_stState.xJumpDetected := TRUE;
        iq_stState.udiRejectedJumpCount :=
            iq_stState.udiRejectedJumpCount + UDINT#1;

        iq_stState.eStatus := CHANNEL_STATUS_COUNTER_JUMP;

    END_IF;

END_IF;

          
END_FUNCTION_BLOCK

FUNCTION_BLOCK FB_InputFilter
VAR_INPUT
    i_xRaw     : BOOL; // Необработанный дискретный сигнал физического входа.
    i_tOnDelay : TIME; // Минимальное время непрерывного сигнала TRUE.
END_VAR

VAR_OUTPUT
    q_xFiltered : BOOL; // Отфильтрованный сигнал без коротких импульсов и дребезга.
END_VAR

VAR
    fbOnDelay : TON; // Стандартный таймер подтверждения входного сигнала.
END_VAR

            fbOnDelay(
    IN := i_xRaw,
    PT := i_tOnDelay
);

q_xFiltered := fbOnDelay.Q;

          
END_FUNCTION_BLOCK

FUNCTION_BLOCK FB_LineMeter
VAR_INPUT
    i_udiPulseDelta           : UDINT; // Новые импульсы шестого энкодера за цикл ПЛК.
    i_xPulseDataValid         : BOOL;  // TRUE, если приращение разрешено учитывать.
    i_udiPulsesPerRevolution  : UDINT; // Импульсов энкодера за один оборот.
    i_udiWheelCircumferenceMm : UDINT; // Окружность мерного колеса в миллиметрах.
    i_tSpeedSample            : TIME;  // Интервал расчёта скорости линии.
END_VAR

VAR_IN_OUT
    iq_stState : ST_LineState; // Общий метраж и скорость линии.
END_VAR

VAR
    fbSpeedSample       : TON;   // Таймер периодического расчёта скорости.
    uliWindowPulses     : ULINT; // Импульсы за текущий интервал скорости.
    uliWindowLengthMm   : ULINT; // Перемещение за интервал скорости, мм.
    uliTotalLengthValue : ULINT; // Промежуточный расчёт общего метража.
    udiSampleTimeMs     : UDINT; // Интервал скорости в миллисекундах.
END_VAR

            iq_stState.xConfigFault :=
    (i_udiPulsesPerRevolution = UDINT#0)
    OR (i_udiWheelCircumferenceMm = UDINT#0)
    OR (i_tSpeedSample <= T#0ms);


// Накапливаем общий метраж и окно скорости только по исправным данным.
IF i_xPulseDataValid AND NOT iq_stState.xConfigFault THEN

    iq_stState.uliTotalPulses :=
        iq_stState.uliTotalPulses
        + UDINT_TO_ULINT(i_udiPulseDelta);

    uliWindowPulses :=
        uliWindowPulses
        + UDINT_TO_ULINT(i_udiPulseDelta);


    uliTotalLengthValue :=
        iq_stState.uliTotalPulses
        * UDINT_TO_ULINT(i_udiWheelCircumferenceMm);

    iq_stState.uliTotalLengthMm :=
        uliTotalLengthValue
        / UDINT_TO_ULINT(i_udiPulsesPerRevolution);

END_IF;


// Самоперезапускающийся таймер выдаёт импульс примерно раз в i_tSpeedSample.
fbSpeedSample(
    IN := NOT fbSpeedSample.Q,
    PT := i_tSpeedSample
);


IF fbSpeedSample.Q THEN

    IF NOT iq_stState.xConfigFault AND i_xPulseDataValid THEN

        uliWindowLengthMm :=
            (
                uliWindowPulses
                * UDINT_TO_ULINT(i_udiWheelCircumferenceMm)
            )
            / UDINT_TO_ULINT(i_udiPulsesPerRevolution);

        udiSampleTimeMs := TIME_TO_UDINT(i_tSpeedSample);


        // мм * 60 / мс = метров в минуту.
        iq_stState.rSpeedMPerMin :=
            ULINT_TO_REAL(uliWindowLengthMm)
            * 60.0
            / UDINT_TO_REAL(udiSampleTimeMs);

        iq_stState.xMoving := uliWindowPulses > ULINT#0;

    ELSE

        iq_stState.rSpeedMPerMin := 0.0;
        iq_stState.xMoving := FALSE;

    END_IF;


    uliWindowPulses := ULINT#0;

END_IF;

          
END_FUNCTION_BLOCK

FUNCTION_BLOCK FB_RollCounter
VAR_INPUT
    i_udiPulseDelta             : UDINT; // Новые импульсы этого раската за цикл ПЛК.
    i_xPulseDataValid           : BOOL;  // TRUE, если приращение разрешено учитывать.
    i_xSplice                   : BOOL;  // Отфильтрованная команда SPLICE.
    i_xReset                    : BOOL;  // Отфильтрованная команда ручного RESET.
    i_udiPulsesPerRevolution    : UDINT; // Импульсов энкодера за один оборот.
    i_udiWheelCircumferenceMm   : UDINT; // Окружность мерного колеса в миллиметрах.
    i_uliManualResetMinLengthMm : ULINT; // Минимальная длина для учёта ручного RESET.
END_VAR

VAR_IN_OUT
    iq_stState : ST_RollState; // Состояние конкретного раската.
END_VAR

VAR
    xPreviousSplice : BOOL;  // Уровень SPLICE на предыдущем цикле.
    xPreviousReset  : BOOL;  // Уровень RESET на предыдущем цикле.
    xSpliceRising   : BOOL;  // Одноцикловый фронт SPLICE.
    xResetRising    : BOOL;  // Одноцикловый фронт RESET.
    xCommandsArmed  : BOOL;  // Команды разрешены после первого отпускания обеих кнопок.
    uliLengthValue  : ULINT; // Промежуточный расчёт длины в миллиметрах.
END_VAR

            // Эти признаки активны только один цикл программы.
iq_stState.xRollCompleted := FALSE;
iq_stState.xShortResetDiscarded := FALSE;
xSpliceRising := FALSE;
xResetRising := FALSE;


// После запуска обе кнопки должны хотя бы один раз быть отпущены.
// Это не позволяет зажатой кнопке завершить рулон при старте ПЛК.
IF NOT xCommandsArmed THEN

    IF NOT i_xSplice AND NOT i_xReset THEN
        xCommandsArmed := TRUE;
    END_IF;

ELSE

    xSpliceRising := i_xSplice AND NOT xPreviousSplice;
    xResetRising := i_xReset AND NOT xPreviousReset;

END_IF;


// Проверяем параметры пересчёта.
iq_stState.xConfigFault :=
    (i_udiPulsesPerRevolution = UDINT#0)
    OR (i_udiWheelCircumferenceMm = UDINT#0);


// Нумерация внутренних рулонов каждого канала начинается с единицы.
IF iq_stState.udiRollSequenceNumber = UDINT#0 THEN
    iq_stState.udiRollSequenceNumber := UDINT#1;
END_IF;


// Накапливаем только достоверное приращение HSC.
IF i_xPulseDataValid AND NOT iq_stState.xConfigFault THEN

    iq_stState.uliCurrentRollPulses :=
        iq_stState.uliCurrentRollPulses
        + UDINT_TO_ULINT(i_udiPulseDelta);


    // импульсы * окружность / импульсов на оборот = миллиметры
    uliLengthValue :=
        iq_stState.uliCurrentRollPulses
        * UDINT_TO_ULINT(i_udiWheelCircumferenceMm);

    iq_stState.uliCurrentLengthMm :=
        uliLengthValue
        / UDINT_TO_ULINT(i_udiPulsesPerRevolution);

END_IF;


// SPLICE всегда завершает рулон.
// RESET завершает рулон только при достижении установленного порога.
IF NOT iq_stState.xConfigFault
   AND
   (
       xSpliceRising
       OR
       (
           xResetRising
           AND
           (iq_stState.uliCurrentLengthMm >= i_uliManualResetMinLengthMm)
       )
   ) THEN

    iq_stState.uliPreviousRollPulses :=
        iq_stState.uliCurrentRollPulses;

    iq_stState.uliPreviousRollLengthMm :=
        iq_stState.uliCurrentLengthMm;


    iq_stState.uliCurrentRollPulses := ULINT#0;
    iq_stState.uliCurrentLengthMm := ULINT#0;


    IF iq_stState.udiRollSequenceNumber < UDINT#4294967295 THEN
        iq_stState.udiRollSequenceNumber :=
            iq_stState.udiRollSequenceNumber + UDINT#1;
    ELSE
        iq_stState.udiRollSequenceNumber := UDINT#1;
    END_IF;


    IF xSpliceRising THEN
        iq_stState.eLastEndReason := ROLL_END_SPLICE;
    ELSE
        iq_stState.eLastEndReason := ROLL_END_RESET;
    END_IF;


    iq_stState.xRollCompleted := TRUE;


// Короткий ручной RESET очищает только текущий рулон.
// Предыдущий учтённый рулон и номер последовательности не изменяются.
ELSIF NOT iq_stState.xConfigFault AND xResetRising THEN

    iq_stState.uliLastDiscardedLengthMm :=
        iq_stState.uliCurrentLengthMm;

    iq_stState.uliDiscardedTotalLengthMm :=
        iq_stState.uliDiscardedTotalLengthMm
        + iq_stState.uliCurrentLengthMm;

    iq_stState.uliCurrentRollPulses := ULINT#0;
    iq_stState.uliCurrentLengthMm := ULINT#0;
    iq_stState.xShortResetDiscarded := TRUE;

END_IF;


// Запоминаем уровни кнопок для обнаружения следующего фронта.
xPreviousSplice := i_xSplice;
xPreviousReset := i_xReset;

          
END_FUNCTION_BLOCK

FUNCTION_BLOCK FB_RollEventQueue
VAR_INPUT
    i_a_xEnqueue       : ARRAY[1..5] OF BOOL;         // Одноцикловые запросы добавления от пяти раскатов.
    i_a_stEvent        : ARRAY[1..5] OF ST_RollEvent; // Данные новых событий; EventId назначит очередь.
    i_udiAckEventId    : UDINT;                       // EventId, подтверждённый службой после записи в SQLite.
    i_wAckCommand      : WORD;                        // Команда 16#A55A подтверждает готовность AckEventId.
END_VAR

VAR_IN_OUT
    iq_a_stQueue        : ARRAY[0..127] OF ST_RollEvent; // Постоянный массив событий из PersistentVars.
    iq_uiQueueHead      : UINT;                          // Индекс первого события очереди.
    iq_uiQueueTail      : UINT;                          // Индекс следующей свободной ячейки.
    iq_uiQueueCount     : UINT;                          // Количество событий в очереди.
    iq_udiNextEventId   : UDINT;                         // Следующий уникальный EventId.
    iq_udiOverflowCount : UDINT;                         // Счётчик событий, не попавших в полную очередь.
END_VAR

VAR_OUTPUT
    q_xEventReady        : BOOL;                       // TRUE: на выходе находится событие для сервера.
    q_stCurrentEvent     : ST_RollEvent;               // Первое событие, ожидающее передачи и подтверждения.
    q_uiQueueCount       : UINT;                       // Текущая заполненность очереди для диагностики.
    q_xQueueFull         : BOOL;                       // TRUE: заняты все 128 ячеек.
    q_xStorageFault      : BOOL;                       // Повреждены индексы или счётчик постоянной очереди.
    q_xEventIdExhausted  : BOOL;                       // Достигнут максимальный UDINT EventId.
    q_xAckAccepted       : BOOL;                       // Одноцикловый признак принятого подтверждения.
    q_xAckRejected       : BOOL;                       // Одноцикловый признак неверного подтверждения.
    q_xAckCommandConsumed: BOOL;                       // Требует очистить регистр команды подтверждения.
    q_a_xEnqueued        : ARRAY[1..5] OF BOOL;        // Какие запросы были успешно помещены в очередь.
END_VAR

VAR
    iChannel     : INT;          // Индекс обработки запросов пяти раскатов.
    stEventToAdd : ST_RollEvent; // Копия события перед назначением уникального EventId.
    stEmptyEvent : ST_RollEvent; // Пустое значение выхода, когда очередь не содержит событий.
END_VAR

VAR CONSTANT
    c_uiQueueCapacity : UINT  := UINT#128;                  // Количество ячеек постоянной очереди.
    c_uiLastQueueIndex: UINT  := UINT#127;                  // Последний допустимый индекс массива.
    c_wAckCommand     : WORD  := WORD#16#A55A;              // Защитная команда подтверждения сервера.
    c_udiMaxEventId   : UDINT := UDINT#4294967295;        // Максимальное значение UDINT.
END_VAR

            // Одноцикловые выходы сбрасываются в начале каждого вызова.
q_xAckAccepted := FALSE;
q_xAckRejected := FALSE;
q_xAckCommandConsumed := FALSE;
q_xEventIdExhausted := FALSE;

FOR iChannel := 1 TO 5 DO
    q_a_xEnqueued[iChannel] := FALSE;
END_FOR;


// Проверяем целостность служебных данных, восстановленных после включения ПЛК.
q_xStorageFault :=
    (iq_uiQueueHead > c_uiLastQueueIndex)
    OR (iq_uiQueueTail > c_uiLastQueueIndex)
    OR (iq_uiQueueCount > c_uiQueueCapacity)
    OR (iq_udiNextEventId = UDINT#0);


IF NOT q_xStorageFault THEN

    // Сначала обрабатываем подтверждение, чтобы при полной очереди
    // в этом же цикле освободилось место для нового события.
    IF i_wAckCommand = c_wAckCommand THEN

        q_xAckCommandConsumed := TRUE;

        IF (iq_uiQueueCount > UINT#0)
           AND (iq_a_stQueue[iq_uiQueueHead].udiEventId = i_udiAckEventId) THEN

            IF iq_uiQueueHead >= c_uiLastQueueIndex THEN
                iq_uiQueueHead := UINT#0;
            ELSE
                iq_uiQueueHead := iq_uiQueueHead + UINT#1;
            END_IF;

            iq_uiQueueCount := iq_uiQueueCount - UINT#1;
            q_xAckAccepted := TRUE;

        ELSE

            // Очередь пустая либо сервер подтвердил не текущее событие.
            q_xAckRejected := TRUE;

        END_IF;

    END_IF;


    // За один цикл могут одновременно завершиться несколько раскатов.
    FOR iChannel := 1 TO 5 DO

        IF i_a_xEnqueue[iChannel] THEN

            IF (iq_uiQueueCount < c_uiQueueCapacity)
               AND (iq_udiNextEventId < c_udiMaxEventId) THEN

                stEventToAdd := i_a_stEvent[iChannel];
                stEventToAdd.udiEventId := iq_udiNextEventId;

                iq_a_stQueue[iq_uiQueueTail] := stEventToAdd;

                IF iq_uiQueueTail >= c_uiLastQueueIndex THEN
                    iq_uiQueueTail := UINT#0;
                ELSE
                    iq_uiQueueTail := iq_uiQueueTail + UINT#1;
                END_IF;

                iq_uiQueueCount := iq_uiQueueCount + UINT#1;
                iq_udiNextEventId := iq_udiNextEventId + UDINT#1;
                q_a_xEnqueued[iChannel] := TRUE;

            ELSIF iq_udiNextEventId >= c_udiMaxEventId THEN

                // Теоретическая защита; в реальной эксплуатации этот предел недостижим.
                q_xEventIdExhausted := TRUE;

            ELSE

                // Очередь заполнена: событие не перезаписывает более старые данные.
                IF iq_udiOverflowCount < UDINT#4294967295 THEN
                    iq_udiOverflowCount := iq_udiOverflowCount + UDINT#1;
                END_IF;

            END_IF;

        END_IF;

    END_FOR;

END_IF;


// Сервер всегда видит только первое неподтверждённое событие.
q_uiQueueCount := iq_uiQueueCount;
q_xQueueFull := iq_uiQueueCount >= c_uiQueueCapacity;
q_xEventReady := (iq_uiQueueCount > UINT#0) AND NOT q_xStorageFault;

IF q_xEventReady THEN
    q_stCurrentEvent := iq_a_stQueue[iq_uiQueueHead];
ELSE
    q_stCurrentEvent := stEmptyEvent;
END_IF;

          
END_FUNCTION_BLOCK

FUNCTION_BLOCK FB_ShiftManager
VAR_INPUT
    i_usiShift1StartHour    : USINT; // Начало первой смены, час 0...23.
    i_usiShift2StartHour    : USINT; // Начало второй смены, час 0...23.
    i_udiUtcOffsetSeconds   : UDINT; // Смещение местного времени относительно UTC в секундах.
END_VAR

VAR_IN_OUT
    iq_stState : ST_ShiftState; // Номер смены и диагностические данные RTC.
END_VAR

VAR
    diUtcTimestamp      : DINT;  // Время RTC в секундах с 01.01.1970 UTC; тип функции GetRtc.
    udiUtcTimestamp     : UDINT; // То же время в беззнаковом формате для арифметики.
    udiLocalTimestamp   : UDINT; // UNIX-время после добавления местного смещения.
    udiLocalSecondsDay  : UDINT; // Местное число секунд от начала суток.
    udiDaysRemaining    : UDINT; // Полные дни от 01.01.1970 для расчёта календарной даты.
    usiNewShift         : USINT; // Рассчитанный номер смены.
    uiYear              : UINT;  // Промежуточный год.
    uiMonth             : UINT;  // Промежуточный месяц.
    uiDaysInYear        : UINT;  // Число дней в рассматриваемом году.
    uiDaysInMonth       : UINT;  // Число дней в рассматриваемом месяце.
    xLeapYear           : BOOL;  // TRUE для високосного года.
END_VAR

            iq_stState.xShiftChanged := FALSE;


// GetRtc входит в уже подключённую библиотеку M241 PLCSystem.
// В текущем проекте пространство имён этой библиотеки — SEC.
diUtcTimestamp := SEC.GetRtc();


IF (diUtcTimestamp > DINT#0)
   AND (i_usiShift1StartHour < USINT#24)
   AND (i_usiShift2StartHour < USINT#24)
   AND (i_usiShift1StartHour < i_usiShift2StartHour) THEN

    udiUtcTimestamp := DINT_TO_UDINT(diUtcTimestamp);
    iq_stState.udiTimestampUtc := udiUtcTimestamp;
    iq_stState.udiRtcError := UDINT#0;

    udiLocalTimestamp := udiUtcTimestamp + i_udiUtcOffsetSeconds;
    udiLocalSecondsDay := udiLocalTimestamp MOD UDINT#86400;


    iq_stState.uiLocalHour :=
        UDINT_TO_UINT(udiLocalSecondsDay / UDINT#3600);

    iq_stState.uiLocalMinute :=
        UDINT_TO_UINT(
            (udiLocalSecondsDay MOD UDINT#3600)
            / UDINT#60
        );

    iq_stState.uiLocalSecond :=
        UDINT_TO_UINT(udiLocalSecondsDay MOD UDINT#60);


    // Календарная дата рассчитывается из целого числа дней UNIX-времени.
    // Цикл ограничен текущим диапазоном UDINT и выполняется не более 137 раз.
    udiDaysRemaining := udiLocalTimestamp / UDINT#86400;
    uiYear := UINT#1970;

    xLeapYear :=
        ((uiYear MOD UINT#4) = UINT#0)
        AND
        (
            ((uiYear MOD UINT#100) <> UINT#0)
            OR ((uiYear MOD UINT#400) = UINT#0)
        );
    IF xLeapYear THEN
        uiDaysInYear := UINT#366;
    ELSE
        uiDaysInYear := UINT#365;
    END_IF;

    WHILE udiDaysRemaining >= UINT_TO_UDINT(uiDaysInYear) DO
        udiDaysRemaining :=
            udiDaysRemaining - UINT_TO_UDINT(uiDaysInYear);
        uiYear := uiYear + UINT#1;

        xLeapYear :=
            ((uiYear MOD UINT#4) = UINT#0)
            AND
            (
                ((uiYear MOD UINT#100) <> UINT#0)
                OR ((uiYear MOD UINT#400) = UINT#0)
            );
        IF xLeapYear THEN
            uiDaysInYear := UINT#366;
        ELSE
            uiDaysInYear := UINT#365;
        END_IF;
    END_WHILE;

    uiMonth := UINT#1;
    WHILE uiMonth <= UINT#12 DO
        CASE uiMonth OF
            UINT#2:
                IF xLeapYear THEN
                    uiDaysInMonth := UINT#29;
                ELSE
                    uiDaysInMonth := UINT#28;
                END_IF;
            UINT#4, UINT#6, UINT#9, UINT#11:
                uiDaysInMonth := UINT#30;
            ELSE
                uiDaysInMonth := UINT#31;
        END_CASE;

        IF udiDaysRemaining < UINT_TO_UDINT(uiDaysInMonth) THEN
            EXIT;
        END_IF;

        udiDaysRemaining :=
            udiDaysRemaining - UINT_TO_UDINT(uiDaysInMonth);
        uiMonth := uiMonth + UINT#1;
    END_WHILE;

    iq_stState.uiLocalYear := uiYear;
    iq_stState.uiLocalMonth := uiMonth;
    iq_stState.uiLocalDay := UDINT_TO_UINT(udiDaysRemaining) + UINT#1;


    IF (iq_stState.uiLocalHour >= USINT_TO_UINT(i_usiShift1StartHour))
       AND (iq_stState.uiLocalHour < USINT_TO_UINT(i_usiShift2StartHour)) THEN

        usiNewShift := USINT#1;

    ELSE

        usiNewShift := USINT#2;

    END_IF;


    IF (iq_stState.usiCurrentShift <> USINT#0)
       AND (iq_stState.usiCurrentShift <> usiNewShift) THEN

        iq_stState.xShiftChanged := TRUE;

    END_IF;


    iq_stState.usiCurrentShift := usiNewShift;
    iq_stState.xRtcValid := TRUE;


ELSE

    iq_stState.xRtcValid := FALSE;
    iq_stState.usiCurrentShift := USINT#0;
    iq_stState.uiLocalHour := UINT#0;
    iq_stState.uiLocalMinute := UINT#0;
    iq_stState.uiLocalSecond := UINT#0;
    iq_stState.uiLocalYear := UINT#0;
    iq_stState.uiLocalMonth := UINT#0;
    iq_stState.uiLocalDay := UINT#0;
    iq_stState.udiTimestampUtc := UDINT#0;

    // 1 означает, что RTC ещё не содержит корректного UNIX-времени.
    IF diUtcTimestamp <= DINT#0 THEN
        iq_stState.udiRtcError := UDINT#1;
    ELSE
        // Максимальное значение означает ошибку настройки границ смен.
        iq_stState.udiRtcError := UDINT#4294967295;
    END_IF;

END_IF;

          
END_FUNCTION_BLOCK

FUNCTION_BLOCK FB_StopJournalQueue
VAR_INPUT
    i_a_xEnqueue   : ARRAY[1..2] OF BOOL; // 1=граница смены, 2=переход состояния/заказ.
    i_a_stEvent    : ARRAY[1..2] OF ST_StopJournalEvent;
    i_udiAckEventId: UDINT;
    i_wAckCommand  : WORD;
END_VAR

VAR_IN_OUT
    iq_a_stQueue    : ARRAY[0..127] OF ST_StopJournalEvent;
    iq_uiHead       : UINT;
    iq_uiTail       : UINT;
    iq_uiCount      : UINT;
    iq_udiNextId    : UDINT;
    iq_udiOverflow  : UDINT;
END_VAR

VAR_OUTPUT
    q_xReady        : BOOL;
    q_stHead        : ST_StopJournalEvent;
    q_xFull         : BOOL;
    q_xStorageFault : BOOL;
    q_xIdExhausted  : BOOL;
    q_xAckConsumed  : BOOL;
    q_xAckAccepted  : BOOL;
    q_xAckRejected  : BOOL;
END_VAR

VAR
    iEvent          : INT;
    stToAdd         : ST_StopJournalEvent;
    stEmpty         : ST_StopJournalEvent;
END_VAR

            q_xAckConsumed := FALSE;
q_xAckAccepted := FALSE;
q_xAckRejected := FALSE;
q_xIdExhausted := FALSE;

q_xStorageFault :=
    (iq_uiHead > UINT#127)
    OR (iq_uiTail > UINT#127)
    OR (iq_uiCount > UINT#128)
    OR (iq_udiNextId = UDINT#0);

IF NOT q_xStorageFault THEN
    // Только подтверждение головы очереди освобождает событие.
    IF i_wAckCommand = WORD#16#A55B THEN
        q_xAckConsumed := TRUE;
        IF (iq_uiCount > UINT#0)
           AND (iq_a_stQueue[iq_uiHead].udiEventId = i_udiAckEventId) THEN
            IF iq_uiHead = UINT#127 THEN
                iq_uiHead := UINT#0;
            ELSE
                iq_uiHead := iq_uiHead + UINT#1;
            END_IF;
            iq_uiCount := iq_uiCount - UINT#1;
            q_xAckAccepted := TRUE;
        ELSE
            q_xAckRejected := TRUE;
        END_IF;
    END_IF;

    FOR iEvent := 1 TO 2 DO
        IF i_a_xEnqueue[iEvent] THEN
            IF (iq_uiCount < UINT#128)
               AND (iq_udiNextId < UDINT#4294967295) THEN
                stToAdd := i_a_stEvent[iEvent];
                stToAdd.udiEventId := iq_udiNextId;
                iq_a_stQueue[iq_uiTail] := stToAdd;
                IF iq_uiTail = UINT#127 THEN
                    iq_uiTail := UINT#0;
                ELSE
                    iq_uiTail := iq_uiTail + UINT#1;
                END_IF;
                iq_uiCount := iq_uiCount + UINT#1;
                iq_udiNextId := iq_udiNextId + UDINT#1;
            ELSIF iq_udiNextId >= UDINT#4294967295 THEN
                q_xIdExhausted := TRUE;
            ELSE
                IF iq_udiOverflow < UDINT#4294967295 THEN
                    iq_udiOverflow := iq_udiOverflow + UDINT#1;
                END_IF;
            END_IF;
        END_IF;
    END_FOR;
END_IF;

q_xFull := iq_uiCount >= UINT#128;
q_xReady := (iq_uiCount > UINT#0) AND NOT q_xStorageFault;
IF q_xReady THEN
    q_stHead := iq_a_stQueue[iq_uiHead];
ELSE
    q_stHead := stEmpty;
END_IF;

          
END_FUNCTION_BLOCK

FUNCTION_BLOCK FB_StopMachine
VAR_INPUT
    i_uliTotalLengthMm               : ULINT; // Общий метраж шестого энкодера.
    i_rSpeedMPerMin                  : REAL;  // Измеренная скорость линии.
    i_xMoving                        : BOOL;  // За последний интервал были импульсы линии.
    i_xLineDataValid                 : BOOL;  // Данные шестого HSC разрешено использовать.
    i_usiCurrentShift                : USINT; // Номер текущей смены 1 или 2.
    i_xShiftChanged                  : BOOL;  // Одноцикловый признак смены.
    i_xRtcValid                      : BOOL;  // Часы ПЛК исправны.
    i_wRestoredState                 : WORD;  // Последняя причина из отдельного постоянного блока.
    i_wCommandCode                   : WORD;  // Код команды HMI.
    i_wCommandSequence               : WORD;  // Новый номер для каждого нажатия.
    i_wParam0                        : WORD;  // Параметр команды 0.
    i_wParam1                        : WORD;  // Параметр команды 1.
    i_wParam2                        : WORD;  // Параметр команды 2.
    i_wSettingStartDetectLengthDm    : WORD;  // Новый порог подтверждения движения, 0,1 м.
    i_wSettingAreaCoefficientX100    : WORD;  // Новый коэффициент площади x 100.
    i_wSettingChangeoverTenthsMin    : WORD;  // Новое время переналадки, 0,1 мин.
    i_wServerOrderCommand            : WORD;  // 16#4F52 применяется после записи всего пакета заказа.
    i_wServerOrderSequence           : WORD;  // Новый номер для каждой записи заказа сервером.
    i_udiServerOrderDatabaseId       : UDINT; // NumZ из базы данных.
    i_udiServerOrderTechnicalCard    : UDINT; // NumTK из базы данных.
    i_udiServerOrderNumber           : UDINT; // Числовая часть Zakaz для отображения.
    i_wServerOrderSourceShift        : WORD;  // NumSM из базы данных.
    i_wServerOrderNominalSpeed       : WORD;  // Efficiency из базы данных.
    i_wServerChangeoverTenthsMin     : WORD;  // ReconfigurationT x 10.
END_VAR

VAR_IN_OUT
    iq_stPersistent : ST_StopMachinePersistent;
    iq_stState      : ST_StopMachineState;
END_VAR

VAR_OUTPUT
    q_xCommandConsumed : BOOL; // PLC принял пакет команды и может очистить CommandCode.
    q_xServerOrderCommandConsumed : BOOL; // PLC обработал/отклонил и может очистить серверную команду.
    q_xBreakRecorded : BOOL; // Приняты подробности обрыва, включая изменение причины в том же состоянии.
END_VAR

VAR
    fbNoFeed                 : TON;
    fbChangeover             : TON;
    uliRunDetectBaselineMm   : ULINT;
    uliOrderDeltaMm          : ULINT;
    uliShiftDeltaMm          : ULINT;
    uliOrderLengthDm         : ULINT;
    uliShiftLengthDm         : ULINT;
    uliOrderAreaX100         : ULINT;
    uliShiftAreaX100         : ULINT;
    udiChangeoverTimeMs      : UDINT;
    udiElapsedMs             : UDINT;
    udiRemainingMs           : UDINT;
    xSettingsValid           : BOOL;
    xBreakRecordedPulse      : BOOL;
END_VAR

            q_xCommandConsumed := FALSE;
q_xServerOrderCommandConsumed := FALSE;
q_xBreakRecorded := FALSE;
xBreakRecordedPulse := FALSE;


// При первом запуске либо после изменения структуры задаём безопасные значения.
IF iq_stPersistent.wConfigSignature <> GVL_Constants.c_wStopMachineSignature THEN
    iq_stPersistent.wConfigSignature := GVL_Constants.c_wStopMachineSignature;
    iq_stPersistent.udiOrderNumber := UDINT#0;
    iq_stPersistent.udiOrderDatabaseId := UDINT#0;
    iq_stPersistent.udiOrderTechnicalCard := UDINT#0;
    iq_stPersistent.uiOrderSourceShift := UINT#0;
    iq_stPersistent.uiOrderNominalSpeed := UINT#0;
    iq_stPersistent.uiOperatorNumber := UINT#0;
    iq_stPersistent.wLastServerOrderSequence := i_wServerOrderSequence;
    iq_stPersistent.uliOrderBaselineMm := i_uliTotalLengthMm;
    iq_stPersistent.uliShiftBaselineMm := i_uliTotalLengthMm;
    iq_stPersistent.uiAreaCoefficientX100 := GVL_Constants.c_uiStopDefaultAreaCoefficientX100;
    iq_stPersistent.uiStartDetectLengthDm := GVL_Constants.c_uiStopDefaultStartDetectLengthDm;
    iq_stPersistent.uiChangeoverSetpointTenthsMin := GVL_Constants.c_uiStopDefaultChangeoverTenthsMin;
    iq_stPersistent.usiLastShiftNumber := i_usiCurrentShift;
END_IF;


IF NOT iq_stState.xInitialized THEN
    // После перезапуска не объявляем работу до импульсов энкодера.
    // Известную ручную причину остановки, если она была, сохраняем.
    IF (i_wRestoredState = GVL_Constants.c_wStopStateStopped)
       OR (i_wRestoredState = GVL_Constants.c_wStopStateNoFeed)
       OR (i_wRestoredState = GVL_Constants.c_wStopStateChangeover)
       OR (i_wRestoredState = GVL_Constants.c_wStopStateProduction)
       OR (i_wRestoredState = GVL_Constants.c_wStopStatePpr)
       OR (i_wRestoredState = GVL_Constants.c_wStopStateLunch)
       OR (i_wRestoredState = GVL_Constants.c_wStopStateRepair)
       OR (i_wRestoredState = GVL_Constants.c_wStopStateAlarm)
       OR (i_wRestoredState = GVL_Constants.c_wStopStateTechnology)
       OR (i_wRestoredState = GVL_Constants.c_wStopStateBreak) THEN
        iq_stState.wStateCode := i_wRestoredState;
    ELSE
        iq_stState.wStateCode := WORD#0; // Пока не определено движение после запуска.
    END_IF;
    iq_stState.wLastCommandResult := GVL_Constants.c_wStopResultNone;
    iq_stState.wLastProcessedSequence := i_wCommandSequence;
    iq_stState.wLastServerOrderResult := WORD#0;
    iq_stState.wLastServerOrderSequence := iq_stPersistent.wLastServerOrderSequence;
    iq_stState.xServerOrderValid := iq_stPersistent.udiOrderDatabaseId <> UDINT#0;
    iq_stState.xPackingComplete := FALSE;
    iq_stState.xCommandRejected := FALSE;
    uliRunDetectBaselineMm := i_uliTotalLengthMm;
    iq_stState.xInitialized := TRUE;
END_IF;


// Заказ может изменить только серверный интерфейс. Сервер пишет параметры,
// затем новый sequence и только после этого команду 16#4F52.
IF i_wServerOrderCommand <> WORD#0 THEN
    q_xServerOrderCommandConsumed := TRUE;

    IF i_wServerOrderSequence <> iq_stPersistent.wLastServerOrderSequence THEN
        iq_stPersistent.wLastServerOrderSequence := i_wServerOrderSequence;
        iq_stState.wLastServerOrderSequence := i_wServerOrderSequence;

        IF i_wServerOrderCommand <> GVL_Constants.c_wServerOrderApplyCommand THEN
            iq_stState.wLastServerOrderResult := WORD#2;
        ELSIF (i_udiServerOrderDatabaseId = UDINT#0)
           OR (i_wServerOrderSourceShift = WORD#0)
           OR (i_wServerChangeoverTenthsMin > WORD#6000) THEN
            iq_stState.wLastServerOrderResult := WORD#3;
        ELSE
            iq_stPersistent.udiOrderDatabaseId := i_udiServerOrderDatabaseId;
            iq_stPersistent.udiOrderTechnicalCard := i_udiServerOrderTechnicalCard;
            iq_stPersistent.udiOrderNumber := i_udiServerOrderNumber;
            iq_stPersistent.uiOrderSourceShift := WORD_TO_UINT(i_wServerOrderSourceShift);
            iq_stPersistent.uiOrderNominalSpeed := WORD_TO_UINT(i_wServerOrderNominalSpeed);
            iq_stPersistent.uiChangeoverSetpointTenthsMin :=
                WORD_TO_UINT(i_wServerChangeoverTenthsMin);
            iq_stPersistent.uliOrderBaselineMm := i_uliTotalLengthMm;

            iq_stState.xPackingComplete := FALSE;
            iq_stState.xServerOrderValid := TRUE;
            iq_stState.wStateCode := GVL_Constants.c_wStopStateChangeover;
            iq_stState.wLastServerOrderResult := WORD#1;
            uliRunDetectBaselineMm := i_uliTotalLengthMm;
        END_IF;
    END_IF;
END_IF;


iq_stState.xConfigFault :=
    (iq_stPersistent.uiAreaCoefficientX100 = UINT#0)
    OR (iq_stPersistent.uiAreaCoefficientX100 > UINT#1000)
    OR (iq_stPersistent.uiStartDetectLengthDm = UINT#0)
    OR (iq_stPersistent.uiStartDetectLengthDm > UINT#6000)
    OR (iq_stPersistent.uiChangeoverSetpointTenthsMin > UINT#6000);


// Сброс аппаратного счётчика не должен создавать отрицательные или огромные дельты.
IF i_uliTotalLengthMm < iq_stPersistent.uliOrderBaselineMm THEN
    iq_stPersistent.uliOrderBaselineMm := i_uliTotalLengthMm;
END_IF;

IF i_uliTotalLengthMm < iq_stPersistent.uliShiftBaselineMm THEN
    iq_stPersistent.uliShiftBaselineMm := i_uliTotalLengthMm;
END_IF;


// Сравнение с постоянным номером смены также ловит смену, прошедшую при
// выключенном PLC, когда однократного xShiftChanged уже не было.
IF ((i_usiCurrentShift = USINT#1) OR (i_usiCurrentShift = USINT#2))
   AND (i_xShiftChanged
        OR (iq_stPersistent.usiLastShiftNumber <> i_usiCurrentShift)) THEN
    iq_stPersistent.uliShiftBaselineMm := i_uliTotalLengthMm;
    iq_stPersistent.usiLastShiftNumber := i_usiCurrentShift;
END_IF;


// Любой ненулевой CommandCode очищается. Действие выполняется только один раз
// при новом sequence, поэтому оставшийся после перезапуска пакет не повторится.
IF i_wCommandCode <> WORD#0 THEN
    q_xCommandConsumed := TRUE;

    IF i_wCommandSequence <> iq_stState.wLastProcessedSequence THEN
        iq_stState.wLastProcessedSequence := i_wCommandSequence;
        iq_stState.wLastCommandResult := GVL_Constants.c_wStopResultAccepted;
        iq_stState.xCommandRejected := FALSE;

        // Причина остановки принимается только при исправном энкодере и
        // отсутствии движения. HMI не может объявить работу без движения.
        IF ((i_wCommandCode = WORD#2)
            AND (NOT i_xMoving OR NOT i_xLineDataValid))
           OR (((i_wCommandCode = WORD#1)
                OR ((i_wCommandCode >= WORD#3) AND (i_wCommandCode <= WORD#10)))
               AND (i_xMoving OR NOT i_xLineDataValid)) THEN
            iq_stState.wLastCommandResult := GVL_Constants.c_wStopResultInvalidState;
            iq_stState.xCommandRejected := TRUE;
        ELSE
        CASE i_wCommandCode OF

        1: // СТОП: меняет только состояние линии в отчёте.
            iq_stState.wStateCode := GVL_Constants.c_wStopStateStopped;
            uliRunDetectBaselineMm := i_uliTotalLengthMm;

        2: // ПУСК: меняет только состояние линии в отчёте.
            iq_stState.wStateCode := GVL_Constants.c_wStopStateRunning;

        3: // ПЕРЕНАЛАДКА. Заказ задаёт только сервер; HMI меняет лишь состояние.
            iq_stState.xPackingComplete := FALSE;
            iq_stState.wStateCode := GVL_Constants.c_wStopStateChangeover;
            uliRunDetectBaselineMm := i_uliTotalLengthMm;

        4: // ПРОИЗВОДСТВО
            iq_stState.wStateCode := GVL_Constants.c_wStopStateProduction;
            uliRunDetectBaselineMm := i_uliTotalLengthMm;

        5: // ОБЕД
            iq_stState.wStateCode := GVL_Constants.c_wStopStateLunch;
            uliRunDetectBaselineMm := i_uliTotalLengthMm;

        6: // ППР
            iq_stState.wStateCode := GVL_Constants.c_wStopStatePpr;
            uliRunDetectBaselineMm := i_uliTotalLengthMm;

        7: // РЕМОНТ
            iq_stState.wStateCode := GVL_Constants.c_wStopStateRepair;
            uliRunDetectBaselineMm := i_uliTotalLengthMm;

        8: // АВАРИЯ
            iq_stState.wStateCode := GVL_Constants.c_wStopStateAlarm;
            uliRunDetectBaselineMm := i_uliTotalLengthMm;

        9: // ТЕХНОЛОГИЯ
            iq_stState.wStateCode := GVL_Constants.c_wStopStateTechnology;
            uliRunDetectBaselineMm := i_uliTotalLengthMm;

        10: // ОБРЫВ: точка 1...5, сторона 1...2, причина 1...3.
            IF (i_wParam0 >= WORD#1) AND (i_wParam0 <= WORD#5)
               AND (i_wParam1 >= WORD#1) AND (i_wParam1 <= WORD#2)
               AND (i_wParam2 >= WORD#1) AND (i_wParam2 <= WORD#3) THEN
                iq_stState.usiLastBreakPoint := WORD_TO_USINT(i_wParam0);
                iq_stState.usiLastBreakSide := WORD_TO_USINT(i_wParam1);
                iq_stState.usiLastBreakReason := WORD_TO_USINT(i_wParam2);
                iq_stState.wStateCode := GVL_Constants.c_wStopStateBreak;
                uliRunDetectBaselineMm := i_uliTotalLengthMm;
                xBreakRecordedPulse := TRUE;
                q_xBreakRecorded := TRUE;
            ELSE
                iq_stState.wLastCommandResult := GVL_Constants.c_wStopResultInvalidParameter;
                iq_stState.xCommandRejected := TRUE;
            END_IF;

        11: // УПАКОВКА ЗАВЕРШЕНА
            iq_stState.xPackingComplete := TRUE;

        12: // НОМЕР ОПЕРАТОРА. Param0=0 выполняет выход пользователя.
            iq_stPersistent.uiOperatorNumber := WORD_TO_UINT(i_wParam0);

        20: // ПРИМЕНИТЬ НАСТРОЙКИ одним атомарным пакетом.
            xSettingsValid :=
                (i_wSettingStartDetectLengthDm >= WORD#1)
                AND (i_wSettingStartDetectLengthDm <= WORD#6000)
                AND (i_wSettingAreaCoefficientX100 >= WORD#1)
                AND (i_wSettingAreaCoefficientX100 <= WORD#1000)
                AND (i_wSettingChangeoverTenthsMin <= WORD#6000);

            IF xSettingsValid THEN
                iq_stPersistent.uiStartDetectLengthDm := WORD_TO_UINT(i_wSettingStartDetectLengthDm);
                iq_stPersistent.uiAreaCoefficientX100 := WORD_TO_UINT(i_wSettingAreaCoefficientX100);
                iq_stPersistent.uiChangeoverSetpointTenthsMin := WORD_TO_UINT(i_wSettingChangeoverTenthsMin);
            ELSE
                iq_stState.wLastCommandResult := GVL_Constants.c_wStopResultInvalidParameter;
                iq_stState.xCommandRejected := TRUE;
            END_IF;

            ELSE
                iq_stState.wLastCommandResult := GVL_Constants.c_wStopResultInvalidCode;
                iq_stState.xCommandRejected := TRUE;

        END_CASE;
        END_IF;
    END_IF;
END_IF;


// Достоверное движение шестого энкодера возвращает статус RUNNING.
// xMoving обновляется раз в секунду; старый порог 50 м здесь не используется.
IF i_xMoving
   AND i_xLineDataValid
   AND NOT iq_stState.xConfigFault
   AND (iq_stState.wStateCode <> GVL_Constants.c_wStopStateRunning) THEN
    iq_stState.wStateCode := GVL_Constants.c_wStopStateRunning;
END_IF;


// Если подтверждённая работа прекратилась, после задержки фиксируем отсутствие подачи.
fbNoFeed(
    IN := ((iq_stState.wStateCode = GVL_Constants.c_wStopStateRunning)
           OR (iq_stState.wStateCode = WORD#0))
          AND i_xLineDataValid
          AND NOT i_xMoving,
    PT := GVL_Constants.c_tStopNoFeedDelay
);

IF fbNoFeed.Q THEN
    iq_stState.wStateCode := GVL_Constants.c_wStopStateNoFeed;
    uliRunDetectBaselineMm := i_uliTotalLengthMm;
END_IF;


// Таймер переналадки. Нулевое задание означает, что контроль времени отключён.
udiChangeoverTimeMs :=
    UINT_TO_UDINT(iq_stPersistent.uiChangeoverSetpointTenthsMin)
    * UDINT#6000;

fbChangeover(
    IN := (iq_stState.wStateCode = GVL_Constants.c_wStopStateChangeover)
          AND (iq_stPersistent.uiChangeoverSetpointTenthsMin > UINT#0),
    PT := UDINT_TO_TIME(udiChangeoverTimeMs)
);

iq_stState.xChangeoverOverdue := fbChangeover.Q;

IF (iq_stState.wStateCode = GVL_Constants.c_wStopStateChangeover)
   AND (iq_stPersistent.uiChangeoverSetpointTenthsMin > UINT#0) THEN
    udiElapsedMs := TIME_TO_UDINT(fbChangeover.ET);
    IF udiElapsedMs < udiChangeoverTimeMs THEN
        udiRemainingMs := udiChangeoverTimeMs - udiElapsedMs;
        iq_stState.uiChangeoverRemainingTenthsMin :=
            UDINT_TO_UINT((udiRemainingMs + UDINT#5999) / UDINT#6000);
    ELSE
        iq_stState.uiChangeoverRemainingTenthsMin := UINT#0;
    END_IF;
ELSE
    iq_stState.uiChangeoverRemainingTenthsMin :=
        iq_stPersistent.uiChangeoverSetpointTenthsMin;
END_IF;


// Расчёт выпуска заказа и смены от независимых базовых отметок.
uliOrderDeltaMm := i_uliTotalLengthMm - iq_stPersistent.uliOrderBaselineMm;
uliShiftDeltaMm := i_uliTotalLengthMm - iq_stPersistent.uliShiftBaselineMm;
uliOrderLengthDm := uliOrderDeltaMm / ULINT#100;
uliShiftLengthDm := uliShiftDeltaMm / ULINT#100;

IF uliOrderLengthDm <= ULINT#4294967295 THEN
    iq_stState.udiCurrentOrderLengthDm := ULINT_TO_UDINT(uliOrderLengthDm);
ELSE
    iq_stState.udiCurrentOrderLengthDm := UDINT#4294967295;
END_IF;

IF uliShiftLengthDm <= ULINT#4294967295 THEN
    iq_stState.udiShiftLengthDm := ULINT_TO_UDINT(uliShiftLengthDm);
ELSE
    iq_stState.udiShiftLengthDm := UDINT#4294967295;
END_IF;

uliOrderAreaX100 :=
    uliOrderLengthDm * UINT_TO_ULINT(iq_stPersistent.uiAreaCoefficientX100) / ULINT#10;
uliShiftAreaX100 :=
    uliShiftLengthDm * UINT_TO_ULINT(iq_stPersistent.uiAreaCoefficientX100) / ULINT#10;

IF uliOrderAreaX100 <= ULINT#4294967295 THEN
    iq_stState.udiCurrentOrderAreaX100 := ULINT_TO_UDINT(uliOrderAreaX100);
ELSE
    iq_stState.udiCurrentOrderAreaX100 := UDINT#4294967295;
END_IF;

IF uliShiftAreaX100 <= ULINT#4294967295 THEN
    iq_stState.udiShiftAreaX100 := ULINT_TO_UDINT(uliShiftAreaX100);
ELSE
    iq_stState.udiShiftAreaX100 := UDINT#4294967295;
END_IF;

iq_stState.udiOrderNumber := iq_stPersistent.udiOrderNumber;
iq_stState.udiOrderDatabaseId := iq_stPersistent.udiOrderDatabaseId;
iq_stState.udiOrderTechnicalCard := iq_stPersistent.udiOrderTechnicalCard;
iq_stState.uiOrderSourceShift := iq_stPersistent.uiOrderSourceShift;
iq_stState.uiOrderNominalSpeed := iq_stPersistent.uiOrderNominalSpeed;
iq_stState.uiOperatorNumber := iq_stPersistent.uiOperatorNumber;

IF i_rSpeedMPerMin <= 0.0 THEN
    iq_stState.uiSpeedDmPerMin := UINT#0;
ELSIF i_rSpeedMPerMin >= 6553.5 THEN
    iq_stState.uiSpeedDmPerMin := UINT#65535;
ELSE
    iq_stState.uiSpeedDmPerMin := REAL_TO_UINT(i_rSpeedMPerMin * 10.0);
END_IF;


// Биты состояния предназначены только для индикации и диагностики HMI.
iq_stState.wStatusBits := WORD#16#0001; // bit 0: блок активен.
IF i_xRtcValid THEN
    iq_stState.wStatusBits := iq_stState.wStatusBits OR WORD#16#0002;
END_IF;
IF i_xMoving THEN
    iq_stState.wStatusBits := iq_stState.wStatusBits OR WORD#16#0004;
END_IF;
IF i_xLineDataValid THEN
    iq_stState.wStatusBits := iq_stState.wStatusBits OR WORD#16#0008;
END_IF;
IF iq_stState.xChangeoverOverdue THEN
    iq_stState.wStatusBits := iq_stState.wStatusBits OR WORD#16#0010;
END_IF;
IF iq_stState.xCommandRejected THEN
    iq_stState.wStatusBits := iq_stState.wStatusBits OR WORD#16#0040;
END_IF;
IF NOT iq_stState.xConfigFault THEN
    iq_stState.wStatusBits := iq_stState.wStatusBits OR WORD#16#0080;
END_IF;
IF xBreakRecordedPulse THEN
    iq_stState.wStatusBits := iq_stState.wStatusBits OR WORD#16#0100;
END_IF;
IF iq_stState.xServerOrderValid THEN
    iq_stState.wStatusBits := iq_stState.wStatusBits OR WORD#16#0200;
END_IF;


iq_stState.wAlarmBits := WORD#0;
IF iq_stState.wStateCode = GVL_Constants.c_wStopStateNoFeed THEN
    iq_stState.wAlarmBits := iq_stState.wAlarmBits OR WORD#16#0001;
END_IF;
IF NOT i_xLineDataValid THEN
    iq_stState.wAlarmBits := iq_stState.wAlarmBits OR WORD#16#0002;
END_IF;
IF iq_stState.xChangeoverOverdue THEN
    iq_stState.wAlarmBits := iq_stState.wAlarmBits OR WORD#16#0004;
END_IF;
IF iq_stState.xCommandRejected THEN
    iq_stState.wAlarmBits := iq_stState.wAlarmBits OR WORD#16#0008;
END_IF;
IF iq_stState.xConfigFault THEN
    iq_stState.wAlarmBits := iq_stState.wAlarmBits OR WORD#16#0010;
END_IF;

          
END_FUNCTION_BLOCK

FUNCTION_BLOCK FB_ThreeFlash
VAR_INPUT
    i_xTrigger    : BOOL; // Новый фронт запускает последовательность заново.
    i_tHalfPeriod : TIME; // Длительность жёлтой и обычной полуволн.
END_VAR

VAR_OUTPUT
    q_xFlashOn : BOOL; // TRUE ровно на трёх жёлтых полуволнах.
    q_xActive  : BOOL; // TRUE в течение всей последовательности из шести полуволн.
END_VAR

VAR
    fbPhaseTimer : TON;
    xTriggerPrevious : BOOL;
    xTriggerRising   : BOOL;
    xResetTimer      : BOOL;
    usiPhase         : USINT; // 0 — ожидание; 1...6 — три пары ВКЛ/ВЫКЛ.
END_VAR

            xTriggerRising := i_xTrigger AND NOT xTriggerPrevious;
xTriggerPrevious := i_xTrigger;


// Каждое новое подтверждённое нажатие начинает три вспышки заново.
IF xTriggerRising THEN
    usiPhase := USINT#1;
    xResetTimer := TRUE;
END_IF;


// После каждой полуволны TON сбрасывается на один цикл программы.
IF xResetTimer THEN
    fbPhaseTimer(
        IN := FALSE,
        PT := i_tHalfPeriod
    );
    xResetTimer := FALSE;
ELSE
    fbPhaseTimer(
        IN := usiPhase <> USINT#0,
        PT := i_tHalfPeriod
    );

    IF fbPhaseTimer.Q THEN
        IF usiPhase >= USINT#6 THEN
            usiPhase := USINT#0;
        ELSE
            usiPhase := usiPhase + USINT#1;
        END_IF;
        xResetTimer := TRUE;
    END_IF;
END_IF;


q_xActive := usiPhase <> USINT#0;
q_xFlashOn :=
    (usiPhase = USINT#1)
    OR (usiPhase = USINT#3)
    OR (usiPhase = USINT#5);

          
END_FUNCTION_BLOCK

PROGRAM SR_Main
VAR
    xHscFirstCycle : BOOL := TRUE;                     // Первый цикл: синхронно сбрасывает и запускает шесть HSC.
    a_dwHscRaw     : ARRAY[1..6] OF DWORD;             // Сырые выходы CurrentValue аппаратных HSC.
    iHsc           : INT;                              // Индекс обработки шести HSC.
    iRoll          : INT;                              // Индекс обработки пяти раскатов.
    iDwinWord      : INT;                              // Индекс копирования общей части пакета DWIN.

    a_fbHscTracker     : ARRAY[1..6] OF FB_HscTracker;     // Трекеры приращений шести HSC.
    a_fbSpliceFilter   : ARRAY[1..5] OF FB_InputFilter;    // Фильтры кнопок SPLICE.
    a_fbResetFilter    : ARRAY[1..5] OF FB_InputFilter;    // Фильтры кнопок RESET.
    a_fbRollCounter    : ARRAY[1..5] OF FB_RollCounter;    // Счётчики текущего и предыдущего рулона.
    a_fbDwinDataPacker : ARRAY[1..5] OF FB_DwinDataPacker; // Упаковщики значений для пяти DWIN.
    fbLineMeter        : FB_LineMeter;                     // Скорость и общий метраж шестого энкодера.
    fbShiftManager     : FB_ShiftManager;                  // Определение текущей смены по RTC.
    fbStopMachine      : FB_StopMachine;                   // Изолированная логика Стопмашины линии ЛГК.
    fbStopJournalQueue : FB_StopJournalQueue;              // Независимая постоянная очередь смены состояний ЛГК.
    xStopJournalFirstCycle : BOOL := TRUE;
    a_xStopJournalEnqueue : ARRAY[1..2] OF BOOL;
    a_stStopJournalEnqueue : ARRAY[1..2] OF ST_StopJournalEvent;
    stStopBeforeUpdate : ST_StopMachineState;
    stStopEvent : ST_StopJournalEvent;
    stEmptyStopJournalEvent : ST_StopJournalEvent;
    wStopPreviousState : WORD;
    wStopPreviousShift : WORD;
    udiStopPreviousOrderDbId : UDINT;
    udiStopAckEventId : UDINT;
    iStopJournalPersistentIndex : INT;
    fbInterfaceHeartbeat : TON;                           // Секундный heartbeat интерфейсов HMI.
    a_fbHaiwellActivityTimeout : ARRAY[1..5] OF TON;       // Удержание признака движения между опросами Haiwell.
    a_fbHaiwellResetTimeout    : ARRAY[1..5] OF TON;       // Удержание индикации RESET на Haiwell.
    a_fbHaiwellAttentionFlash  : ARRAY[1..5] OF FB_ThreeFlash; // Три жёлтые вспышки после SPLICE или RESET.
    a_xHaiwellActivitySeen     : ARRAY[1..5] OF BOOL;      // На канале недавно были импульсы.
    a_xHaiwellResetSeen        : ARRAY[1..5] OF BOOL;      // На канале недавно был RESET.

    a_xRollEventRequest  : ARRAY[1..5] OF BOOL;         // Одноцикловые запросы записи завершённых рулонов.
    a_stRollEventRequest : ARRAY[1..5] OF ST_RollEvent; // Данные событий от пяти раскатов до помещения в очередь.
    fbRollEventQueue     : FB_RollEventQueue;            // Постоянная FIFO-очередь событий для службы-сборщика.
    fbEventPacker        : FB_EventPacker;               // Упаковка первого события очереди в 16 Modbus-регистров.
    udiAckEventId        : UDINT;                        // EventId, собранный из двух слов подтверждения сервера.
    iPacketWord          : INT;                          // Индекс копирования 12 слов пакета v2 в GVL_SCADA.
    udiServerOrderDatabaseId    : UDINT;                 // Пакет заказа сервера, собранный из Modbus-слов.
    udiServerOrderTechnicalCard : UDINT;
    udiServerOrderNumber        : UDINT;

    fbCollectorTimeout          : TON;                   // Таймер отсутствия heartbeat службы-сборщика.
    wCollectorHeartbeatPrevious : WORD;                  // Предыдущее значение heartbeat службы-сборщика.
    xCollectorHeartbeatChanged  : BOOL;                  // Одноцикловый признак изменения heartbeat.
    xCollectorHeartbeatSeen     : BOOL;                  // Служба хотя бы один раз изменила heartbeat.
    xCollectorConnected         : BOOL;                  // Heartbeat менялся в течение последних пяти секунд.
    uliHaiwellValueX10          : ULINT;                 // Промежуточное значение длины в 0,1 м.
    udiHaiwellValueX10          : UDINT;                 // Ограниченное 32-битное значение для Modbus.
    uiHaiwellSpeedX10           : UINT;                  // Скорость в 0,1 м/мин.
    uliShiftLengthMm            : ULINT;                 // Промежуточная длина текущей смены, мм.
    uliShiftRawTotalMm          : ULINT;                 // Суммарный расход пяти раскатов за смену, мм.
    udiShiftElapsedSeconds      : UDINT;                 // Прошедшее время текущего сменного интервала.
    rShiftAverageSpeedMPerMin   : REAL;                  // Средняя скорость выпуска с начала сменного интервала.
    xRollPulseThisCycle         : BOOL;                  // За цикл получены достоверные импульсы раската.
    xRollResetThisCycle         : BOOL;                  // За цикл выполнен короткий или учтённый RESET.
    xShiftIntervalExpired       : BOOL;                  // Накопители относятся к прошлому 12-часовому интервалу.
    iPersistentEvent            : INT;                   // Индекс очистки постоянной очереди после смены разметки.
    iPersistentRoll             : INT;                   // Индекс очистки постоянного состояния раскатов.
    stEmptyRollEvent            : ST_RollEvent;          // Нулевой шаблон события для безопасной инициализации.
    stEmptyRollState            : ST_RollState;          // Нулевой шаблон состояния раската.
    stEmptyStopMachine          : ST_StopMachinePersistent; // Нулевой шаблон состояния Стопмашины.
    a_wDwinCommon               : ARRAY[5..12] OF WORD;  // Общие для пяти панелей дата, время, смена и статус RTC.
    a_wDwinRtcCommon            : ARRAY[0..3] OF WORD;   // Команда синхронизации встроенных часов DWIN.
END_VAR

            // ============================================================
// 0. Контроль разметки постоянной памяти
// ============================================================

// При первом запуске этой версии старая PERSISTENT-разметка может содержать
// данные прежнего проекта в новых полях. Несовпадение сигнатуры или версии
// очищает только данные приложения, после чего признак сохраняется.
IF (PersistentVars.dwLayoutSignature <> GVL_Constants.c_dwPersistentLayoutSignature)
   OR (PersistentVars.wLayoutVersion <> GVL_Constants.c_wPersistentLayoutVersion) THEN

    FOR iPersistentEvent := 0 TO 127 DO
        PersistentVars.a_stEventQueue[iPersistentEvent] := stEmptyRollEvent;
    END_FOR;

    FOR iPersistentRoll := 1 TO GVL_Constants.c_iRollChannelCount DO
        PersistentVars.a_stRollState[iPersistentRoll] := stEmptyRollState;
        PersistentVars.a_uliShiftRollPulses[iPersistentRoll] := ULINT#0;
    END_FOR;

    PersistentVars.uiEventQueueHead := UINT#0;
    PersistentVars.uiEventQueueTail := UINT#0;
    PersistentVars.uiEventQueueCount := UINT#0;
    PersistentVars.udiNextEventId := UDINT#1;
    PersistentVars.udiQueueOverflowCount := UDINT#0;
    PersistentVars.stStopMachine := stEmptyStopMachine;
    PersistentVars.usiShiftAccumulatorNumber := USINT#0;
    PersistentVars.udiShiftStartTimestampUtc := UDINT#0;
    PersistentVars.uliShiftOutputPulses := ULINT#0;
    PersistentVars.dwLayoutSignature := GVL_Constants.c_dwPersistentLayoutSignature;
    PersistentVars.wLayoutVersion := GVL_Constants.c_wPersistentLayoutVersion;

END_IF;

// Новый журнал имеет собственную persistent-разметку и не сбрасывает
// существующие счётчики рулонов при первом импорте.
IF PersistentVars.stStopJournal.dwSignature <> DWORD#16#534A4C34 THEN
    FOR iStopJournalPersistentIndex := 0 TO 127 DO
        PersistentVars.stStopJournal.a_stQueue[iStopJournalPersistentIndex] := stEmptyStopJournalEvent;
    END_FOR;
    PersistentVars.stStopJournal.uiHead := UINT#0;
    PersistentVars.stStopJournal.uiTail := UINT#0;
    PersistentVars.stStopJournal.uiCount := UINT#0;
    PersistentVars.stStopJournal.udiNextEventId := UDINT#1;
    PersistentVars.stStopJournal.udiOverflowCount := UDINT#0;
    PersistentVars.stStopJournal.uliLinePulses := ULINT#0;
    PersistentVars.stStopJournal.wLastState := WORD#0;
    PersistentVars.stStopJournal.dwSignature := DWORD#16#534A4C34;
END_IF;

// ============================================================
// 1. Вызов шести аппаратных HSC
// ============================================================

HscSimple_0(
    Enable := TRUE,
    Sync := xHscFirstCycle,
    ACK_Modulo := FALSE,
    HSC_Err => GVL_IO.xHscError[1],
    Validity => GVL_IO.xHscValid[1],
    CurrentValue => a_dwHscRaw[1]
);

HscSimple_1(
    Enable := TRUE,
    Sync := xHscFirstCycle,
    ACK_Modulo := FALSE,
    HSC_Err => GVL_IO.xHscError[2],
    Validity => GVL_IO.xHscValid[2],
    CurrentValue => a_dwHscRaw[2]
);

HscSimple_2(
    Enable := TRUE,
    Sync := xHscFirstCycle,
    ACK_Modulo := FALSE,
    HSC_Err => GVL_IO.xHscError[3],
    Validity => GVL_IO.xHscValid[3],
    CurrentValue => a_dwHscRaw[3]
);

HscSimple_3(
    Enable := TRUE,
    Sync := xHscFirstCycle,
    ACK_Modulo := FALSE,
    HSC_Err => GVL_IO.xHscError[4],
    Validity => GVL_IO.xHscValid[4],
    CurrentValue => a_dwHscRaw[4]
);

HscSimple_4(
    Enable := TRUE,
    Sync := xHscFirstCycle,
    ACK_Modulo := FALSE,
    HSC_Err => GVL_IO.xHscError[5],
    Validity => GVL_IO.xHscValid[5],
    CurrentValue => a_dwHscRaw[5]
);

HscSimple_5(
    Enable := TRUE,
    Sync := xHscFirstCycle,
    ACK_Modulo := FALSE,
    HSC_Err => GVL_IO.xHscError[6],
    Validity => GVL_IO.xHscValid[6],
    CurrentValue => a_dwHscRaw[6]
);


// Sync активен только при первом проходе SR_Main.
xHscFirstCycle := FALSE;


// ============================================================
// 2. Обработка абсолютных значений HSC
// ============================================================

GVL_Diagnostics.stSystem.xAnyHscFault := FALSE;
GVL_Diagnostics.stSystem.xAnyConfigFault := FALSE;


FOR iHsc := 1 TO GVL_Constants.c_iHscChannelCount DO

    GVL_IO.udiHscAbs[iHsc] :=
        DWORD_TO_UDINT(a_dwHscRaw[iHsc]);


    a_fbHscTracker[iHsc](
        i_udiHscAbs := GVL_IO.udiHscAbs[iHsc],
        i_xHscValid := GVL_IO.xHscValid[iHsc],
        i_xHscError := GVL_IO.xHscError[iHsc],
        i_udiCounterRange := GVL_Constants.c_udiHscCounterRange,
        i_udiMaxDeltaPerCycle := GVL_Constants.c_udiMaxPulseDeltaPerCycle,
        iq_stState := GVL_Runtime.a_stHscState[iHsc]
    );


    GVL_Diagnostics.stSystem.a_eHscStatus[iHsc] :=
        GVL_Runtime.a_stHscState[iHsc].eStatus;

    GVL_Diagnostics.stSystem.a_xHscFault[iHsc] :=
        (GVL_Runtime.a_stHscState[iHsc].eStatus <> CHANNEL_STATUS_RUNNING)
        AND
        (GVL_Runtime.a_stHscState[iHsc].eStatus <> CHANNEL_STATUS_STARTING);

    GVL_Diagnostics.stSystem.xAnyHscFault :=
        GVL_Diagnostics.stSystem.xAnyHscFault
        OR GVL_Diagnostics.stSystem.a_xHscFault[iHsc];

    GVL_Diagnostics.stSystem.xAnyConfigFault :=
        GVL_Diagnostics.stSystem.xAnyConfigFault
        OR
        (GVL_Runtime.a_stHscState[iHsc].eStatus = CHANNEL_STATUS_CONFIG_ERROR);

END_FOR;


// ============================================================
// 3. Определение номера текущей смены и времени события
// ============================================================

fbShiftManager(
    i_usiShift1StartHour := GVL_Constants.c_usiShift_1_StartHour,
    i_usiShift2StartHour := GVL_Constants.c_usiShift_2_StartHour,
    i_udiUtcOffsetSeconds := GVL_Constants.c_udiLocalUtcOffsetSeconds,
    iq_stState := GVL_Runtime.stShiftState
);


GVL_Diagnostics.stSystem.xRtcFault :=
    NOT GVL_Runtime.stShiftState.xRtcValid;


// Общая часть пакета всех DWIN. Компоненты времени передаются отдельными
// 16-битными числами, поэтому панели не зависят от порядка слов UDINT.
a_wDwinCommon[5] := UINT_TO_WORD(GVL_Runtime.stShiftState.uiLocalYear);
a_wDwinCommon[6] := UINT_TO_WORD(GVL_Runtime.stShiftState.uiLocalMonth);
a_wDwinCommon[7] := UINT_TO_WORD(GVL_Runtime.stShiftState.uiLocalDay);
a_wDwinCommon[8] := UINT_TO_WORD(GVL_Runtime.stShiftState.uiLocalHour);
a_wDwinCommon[9] := UINT_TO_WORD(GVL_Runtime.stShiftState.uiLocalMinute);
a_wDwinCommon[10] := UINT_TO_WORD(GVL_Runtime.stShiftState.uiLocalSecond);
a_wDwinCommon[11] := USINT_TO_WORD(GVL_Runtime.stShiftState.usiCurrentShift);
IF GVL_Runtime.stShiftState.xRtcValid THEN
    a_wDwinCommon[12] := WORD#1;
ELSE
    a_wDwinCommon[12] := WORD#0;
END_IF;


// Системный RTC DWIN устанавливается записью четырёх слов с VP 009C:
// 5AA5, YYMM, DDHH, MMSS. Год передаётся смещением от 2000.
IF GVL_Runtime.stShiftState.xRtcValid
   AND (GVL_Runtime.stShiftState.uiLocalYear >= UINT#2000)
   AND (GVL_Runtime.stShiftState.uiLocalYear <= UINT#2255)
   AND (GVL_Runtime.stShiftState.uiLocalMonth >= UINT#1)
   AND (GVL_Runtime.stShiftState.uiLocalMonth <= UINT#12)
   AND (GVL_Runtime.stShiftState.uiLocalDay >= UINT#1)
   AND (GVL_Runtime.stShiftState.uiLocalDay <= UINT#31)
   AND (GVL_Runtime.stShiftState.uiLocalHour <= UINT#23)
   AND (GVL_Runtime.stShiftState.uiLocalMinute <= UINT#59)
   AND (GVL_Runtime.stShiftState.uiLocalSecond <= UINT#59) THEN

    a_wDwinRtcCommon[0] := WORD#16#5AA5;
    a_wDwinRtcCommon[1] :=
        SHL(
            UINT_TO_WORD(GVL_Runtime.stShiftState.uiLocalYear - UINT#2000),
            8
        )
        OR UINT_TO_WORD(GVL_Runtime.stShiftState.uiLocalMonth);
    a_wDwinRtcCommon[2] :=
        SHL(UINT_TO_WORD(GVL_Runtime.stShiftState.uiLocalDay), 8)
        OR UINT_TO_WORD(GVL_Runtime.stShiftState.uiLocalHour);
    a_wDwinRtcCommon[3] :=
        SHL(UINT_TO_WORD(GVL_Runtime.stShiftState.uiLocalMinute), 8)
        OR UINT_TO_WORD(GVL_Runtime.stShiftState.uiLocalSecond);

ELSE

    // Нулевая сигнатура запрещает установку DWIN по недостоверному времени.
    a_wDwinRtcCommon[0] := WORD#0;
    a_wDwinRtcCommon[1] := WORD#0;
    a_wDwinRtcCommon[2] := WORD#0;
    a_wDwinRtcCommon[3] := WORD#0;

END_IF;


FOR iDwinWord := 0 TO 3 DO
    GVL_HMI.a_wHmi1RtcSync[iDwinWord] := a_wDwinRtcCommon[iDwinWord];
    GVL_HMI.a_wHmi2RtcSync[iDwinWord] := a_wDwinRtcCommon[iDwinWord];
    GVL_HMI.a_wHmi3RtcSync[iDwinWord] := a_wDwinRtcCommon[iDwinWord];
    GVL_HMI.a_wHmi4RtcSync[iDwinWord] := a_wDwinRtcCommon[iDwinWord];
    GVL_HMI.a_wHmi5RtcSync[iDwinWord] := a_wDwinRtcCommon[iDwinWord];
END_FOR;


// Накопители смены не зависят от сбросов отдельных рулонов. Они используют
// те же проверенные приращения HSC и сохраняются при перезапуске ПЛК.
IF GVL_Runtime.stShiftState.xRtcValid THEN

    xShiftIntervalExpired := FALSE;
    IF PersistentVars.udiShiftStartTimestampUtc <> UDINT#0 THEN
        IF GVL_Runtime.stShiftState.udiTimestampUtc
           < PersistentVars.udiShiftStartTimestampUtc THEN
            xShiftIntervalExpired := TRUE;
        ELSE
            xShiftIntervalExpired :=
                (GVL_Runtime.stShiftState.udiTimestampUtc
                 - PersistentVars.udiShiftStartTimestampUtc)
                >= GVL_Constants.c_udiShiftMaxIntervalSeconds;
        END_IF;
    END_IF;

    IF (PersistentVars.usiShiftAccumulatorNumber < USINT#1)
       OR (PersistentVars.usiShiftAccumulatorNumber > USINT#2)
       OR (PersistentVars.usiShiftAccumulatorNumber <> GVL_Runtime.stShiftState.usiCurrentShift)
       OR (PersistentVars.udiShiftStartTimestampUtc = UDINT#0)
       OR xShiftIntervalExpired THEN

        PersistentVars.usiShiftAccumulatorNumber :=
            GVL_Runtime.stShiftState.usiCurrentShift;
        PersistentVars.udiShiftStartTimestampUtc :=
            GVL_Runtime.stShiftState.udiTimestampUtc;
        PersistentVars.uliShiftOutputPulses := ULINT#0;

        FOR iRoll := 1 TO GVL_Constants.c_iRollChannelCount DO
            PersistentVars.a_uliShiftRollPulses[iRoll] := ULINT#0;
        END_FOR;

    END_IF;

    FOR iRoll := 1 TO GVL_Constants.c_iRollChannelCount DO
        IF GVL_Runtime.a_stHscState[iRoll].xDataValid THEN
            IF PersistentVars.a_uliShiftRollPulses[iRoll]
               <= (ULINT#18446744073709551615
                   - UDINT_TO_ULINT(GVL_Runtime.a_stHscState[iRoll].udiPulseDelta)) THEN
                PersistentVars.a_uliShiftRollPulses[iRoll] :=
                    PersistentVars.a_uliShiftRollPulses[iRoll]
                    + UDINT_TO_ULINT(GVL_Runtime.a_stHscState[iRoll].udiPulseDelta);
            ELSE
                PersistentVars.a_uliShiftRollPulses[iRoll] :=
                    ULINT#18446744073709551615;
                GVL_Diagnostics.stSystem.xAnyConfigFault := TRUE;
            END_IF;
        END_IF;
    END_FOR;

    IF GVL_Runtime.a_stHscState[6].xDataValid THEN
        IF PersistentVars.uliShiftOutputPulses
           <= (ULINT#18446744073709551615
               - UDINT_TO_ULINT(GVL_Runtime.a_stHscState[6].udiPulseDelta)) THEN
            PersistentVars.uliShiftOutputPulses :=
                PersistentVars.uliShiftOutputPulses
                + UDINT_TO_ULINT(GVL_Runtime.a_stHscState[6].udiPulseDelta);
        ELSE
            PersistentVars.uliShiftOutputPulses := ULINT#18446744073709551615;
            GVL_Diagnostics.stSystem.xAnyConfigFault := TRUE;
        END_IF;
    END_IF;

END_IF;


// ============================================================
// 4. Фильтрация кнопок и учёт пяти раскатов
// ============================================================

FOR iRoll := 1 TO GVL_Constants.c_iRollChannelCount DO

    a_fbSpliceFilter[iRoll](
        i_xRaw := GVL_IO.xSplice[iRoll],
        i_tOnDelay := GVL_Constants.c_tInputFilter
    );

    a_fbResetFilter[iRoll](
        i_xRaw := GVL_IO.xReset[iRoll],
        i_tOnDelay := GVL_Constants.c_tInputFilter
    );


    a_fbRollCounter[iRoll](
        i_udiPulseDelta := GVL_Runtime.a_stHscState[iRoll].udiPulseDelta,
        i_xPulseDataValid := GVL_Runtime.a_stHscState[iRoll].xDataValid,
        i_xSplice := a_fbSpliceFilter[iRoll].q_xFiltered,
        i_xReset := a_fbResetFilter[iRoll].q_xFiltered,
        i_udiPulsesPerRevolution := GVL_Constants.c_udiEncoderPulsesPerRevolution,
        i_udiWheelCircumferenceMm := GVL_Constants.c_udiWheelCircumferenceMm,
        i_uliManualResetMinLengthMm := GVL_Constants.c_uliManualResetMinLengthMm,
        iq_stState := PersistentVars.a_stRollState[iRoll]
    );


    GVL_Diagnostics.stSystem.xAnyConfigFault :=
        GVL_Diagnostics.stSystem.xAnyConfigFault
        OR PersistentVars.a_stRollState[iRoll].xConfigFault;


    // При завершении рулона создаём неизменяемый снимок для постоянной очереди.
    a_xRollEventRequest[iRoll] :=
        PersistentVars.a_stRollState[iRoll].xRollCompleted;


    // Одноцикловые признаки преобразуем в устойчивые состояния для HMI,
    // которая опрашивает Modbus значительно медленнее цикла программы ПЛК.
    xRollPulseThisCycle :=
        GVL_Runtime.a_stHscState[iRoll].xDataValid
        AND (GVL_Runtime.a_stHscState[iRoll].udiPulseDelta > UDINT#0);

    IF xRollPulseThisCycle THEN
        a_xHaiwellActivitySeen[iRoll] := TRUE;
    END_IF;

    a_fbHaiwellActivityTimeout[iRoll](
        IN := NOT xRollPulseThisCycle,
        PT := GVL_Constants.c_tHaiwellActivityHold
    );

    IF a_fbHaiwellActivityTimeout[iRoll].Q THEN
        a_xHaiwellActivitySeen[iRoll] := FALSE;
    END_IF;

    xRollResetThisCycle :=
        (
            PersistentVars.a_stRollState[iRoll].xShortResetDiscarded
            OR
            (
                PersistentVars.a_stRollState[iRoll].xRollCompleted
                AND (PersistentVars.a_stRollState[iRoll].eLastEndReason = ROLL_END_RESET)
            )
        );

    IF xRollResetThisCycle THEN
        a_xHaiwellResetSeen[iRoll] := TRUE;
    END_IF;

    a_fbHaiwellResetTimeout[iRoll](
        IN := NOT xRollResetThisCycle,
        PT := GVL_Constants.c_tHaiwellResetHold
    );

    IF a_fbHaiwellResetTimeout[iRoll].Q THEN
        a_xHaiwellResetSeen[iRoll] := FALSE;
    END_IF;

    a_fbHaiwellAttentionFlash[iRoll](
        i_xTrigger := a_fbSpliceFilter[iRoll].q_xFiltered
                      OR a_fbResetFilter[iRoll].q_xFiltered,
        i_tHalfPeriod := GVL_Constants.c_tHaiwellFlashHalfPeriod
    );

    IF a_xRollEventRequest[iRoll] THEN
        a_stRollEventRequest[iRoll].udiEventId := UDINT#0; // Настоящий EventId назначит очередь.
        a_stRollEventRequest[iRoll].udiTimestampUtc := GVL_Runtime.stShiftState.udiTimestampUtc;
        a_stRollEventRequest[iRoll].usiUnwindNumber := INT_TO_USINT(iRoll);
        a_stRollEventRequest[iRoll].usiShiftNumber := GVL_Runtime.stShiftState.usiCurrentShift;
        a_stRollEventRequest[iRoll].eEndReason := PersistentVars.a_stRollState[iRoll].eLastEndReason;

        // Физически недостижимый предел защищает явное преобразование ULINT -> UDINT.
        IF PersistentVars.a_stRollState[iRoll].uliPreviousRollLengthMm <= ULINT#4294967295 THEN
            a_stRollEventRequest[iRoll].udiLengthMm :=
                ULINT_TO_UDINT(PersistentVars.a_stRollState[iRoll].uliPreviousRollLengthMm);
        ELSE
            a_stRollEventRequest[iRoll].udiLengthMm := UDINT#4294967295;
            GVL_Diagnostics.stSystem.xAnyConfigFault := TRUE;
        END_IF;
    END_IF;


    // Подготавливаем индивидуальную часть пакета VP 2000...2004 для своей панели.
    a_fbDwinDataPacker[iRoll](
        i_uliCurrentLengthMm := PersistentVars.a_stRollState[iRoll].uliCurrentLengthMm,
        i_uliPreviousLengthMm := PersistentVars.a_stRollState[iRoll].uliPreviousRollLengthMm,
        i_usiUnwindNumber := INT_TO_USINT(iRoll)
    );


    GVL_Diagnostics.stSystem.a_xHmiOverflow[iRoll] :=
        a_fbDwinDataPacker[iRoll].q_xOverflow;


    // Каждая панель имеет собственный массив, удобный для I/O Mapping.
    CASE iRoll OF

        1:
            GVL_HMI.a_wHmi1Tx[0] := a_fbDwinDataPacker[iRoll].q_wCurrentHigh;
            GVL_HMI.a_wHmi1Tx[1] := a_fbDwinDataPacker[iRoll].q_wCurrentLow;
            GVL_HMI.a_wHmi1Tx[2] := a_fbDwinDataPacker[iRoll].q_wPreviousHigh;
            GVL_HMI.a_wHmi1Tx[3] := a_fbDwinDataPacker[iRoll].q_wPreviousLow;
            GVL_HMI.a_wHmi1Tx[4] := a_fbDwinDataPacker[iRoll].q_wUnwindNumber;
            FOR iDwinWord := 5 TO 12 DO
                GVL_HMI.a_wHmi1Tx[iDwinWord] := a_wDwinCommon[iDwinWord];
            END_FOR;

